   1:  PR[GP1:91,2] = PR[GP1:90,2] + 24.586;
   1:L PR[91] 10mm/sec CNT100;
   1:  PR[GP1:91,1] = PR[GP1:90,1] + 8.241;
   1:  PR[GP1:91,2] = PR[GP1:90,2] + 23.035;
   1:L PR[91] 10mm/sec CNT100;
   1:  PR[GP1:91,1] = PR[GP1:90,1] + 4.572;
   1:  PR[GP1:91,2] = PR[GP1:90,2] + 17.187;
   1:L PR[91] 10mm/sec CNT100;
   1:  PR[GP1:91,1] = PR[GP1:90,1] + 2.350;
   1:  PR[GP1:91,2] = PR[GP1:90,2] + 14.091;
   1:L PR[91] 10mm/sec CNT100;
   1:  PR[GP1:91,1] = PR[GP1:90,1] + -2.900;
   1:L PR[91] 10mm/sec CNT100;
   1:  PR[GP1:91,1] = PR[GP1:90,1] + -6.756;
   1:  PR[GP1:91,2] = PR[GP1:90,2] + 20.165;
   1:L PR[91] 10mm/sec CNT100;
   1:  PR[GP1:91,1] = PR[GP1:90,1] + -8.743;
   1:  PR[GP1:91,2] = PR[GP1:90,2] + 23.019;
   1:L PR[91] 10mm/sec CNT100;
   1:  PR[GP1:91,1] = PR[GP1:90,1] + -10.484;
   1:  PR[GP1:91,2] = PR[GP1:90,2] + 24.588;
   1:L PR[91] 10mm/sec CNT100;
   1:  PR[GP1:91,1] = PR[GP1:90,1] + -18.525;
   1:  PR[GP1:91,2] = PR[GP1:90,2] + 30.630;
   1:L PR[91] 10mm/sec CNT100;
   1:  PR[GP1:91,1] = PR[GP1:90,1] + -19.030;
   1:  PR[GP1:91,2] = PR[GP1:90,2] + 30.917;
   1:L PR[91] 10mm/sec CNT100;
   1:  PR[GP1:91,1] = PR[GP1:90,1] + -21.878;
   1:  PR[GP1:91,2] = PR[GP1:90,2] + 31.816;
   1:L PR[91] 10mm/sec CNT100;
   1:  PR[GP1:91,1] = PR[GP1:90,1] + -30.388;
   1:  PR[GP1:91,2] = PR[GP1:90,2] + 34.743;
   1:L PR[91] 10mm/sec CNT100;
   1:  PR[GP1:91,1] = PR[GP1:90,1] + -33.292;
   1:  PR[GP1:91,2] = PR[GP1:90,2] + 34.868;
   1:L PR[91] 10mm/sec CNT100;
   1:  PR[GP1:91,1] = PR[GP1:90,1] + -42.531;
   1:  PR[GP1:91,2] = PR[GP1:90,2] + 34.793;
   1:L PR[91] 10mm/sec CNT100;
   1:  PR[GP1:91,1] = PR[GP1:90,1] + -48.692;
   1:  PR[GP1:91,2] = PR[GP1:90,2] + 32.836;
   1:L PR[91] 10mm/sec CNT100;
   1:  PR[GP1:91,1] = PR[GP1:90,1] + -54.219;
   1:  PR[GP1:91,2] = PR[GP1:90,2] + 30.834;
   1:L PR[91] 10mm/sec CNT100;
   1:  PR[GP1:91,1] = PR[GP1:90,1] + -61.326;
   1:  PR[GP1:91,2] = PR[GP1:90,2] + 25.314;
   1:L PR[91] 10mm/sec CNT100;
   1:  PR[GP1:91,1] = PR[GP1:90,1] + -63.971;
   1:  PR[GP1:91,2] = PR[GP1:90,2] + 23.133;
   1:L PR[91] 10mm/sec CNT100;
   1:  PR[GP1:91,1] = PR[GP1:90,1] + -69.432;
   1:  PR[GP1:91,2] = PR[GP1:90,2] + 14.214;
   1:L PR[91] 10mm/sec CNT100;
   1:  PR[GP1:91,1] = PR[GP1:90,1] + -70.446;
   1:  PR[GP1:91,2] = PR[GP1:90,2] + 12.486;
   1:L PR[91] 10mm/sec CNT100;
   1:  PR[GP1:91,1] = PR[GP1:90,1] + -72.467;
   1:  PR[GP1:91,2] = PR[GP1:90,2] + 1.672;
   1:L PR[91] 10mm/sec CNT100;
   1:  PR[GP1:91,1] = PR[GP1:90,1] + -72.701;
   1:  PR[GP1:91,2] = PR[GP1:90,2] + 0.583;
   1:L PR[91] 10mm/sec CNT100;
   1:  PR[GP1:91,1] = PR[GP1:90,1] + -72.755;
   1:  PR[GP1:91,2] = PR[GP1:90,2] + 0.282;
   1:L PR[91] 10mm/sec CNT100;
   1:  PR[GP1:91,1] = PR[GP1:90,1] + -70.738;
   1:  PR[GP1:91,2] = PR[GP1:90,2] + -10.290;
   1:L PR[91] 10mm/sec CNT100;
   1:  PR[GP1:91,1] = PR[GP1:90,1] + -70.445;
   1:  PR[GP1:91,2] = PR[GP1:90,2] + -11.930;
   1:L PR[91] 10mm/sec CNT100;
   1:  PR[GP1:91,1] = PR[GP1:90,1] + -69.432;
   1:  PR[GP1:91,2] = PR[GP1:90,2] + -13.656;
   1:L PR[91] 10mm/sec CNT100;
   1:  PR[GP1:91,1] = PR[GP1:90,1] + -63.971;
   1:  PR[GP1:91,2] = PR[GP1:90,2] + -22.575;
   1:L PR[91] 10mm/sec CNT100;
   1:  PR[GP1:91,1] = PR[GP1:90,1] + -61.326;
   1:  PR[GP1:91,2] = PR[GP1:90,2] + -24.756;
   1:L PR[91] 10mm/sec CNT100;
   1:  PR[GP1:91,1] = PR[GP1:90,1] + -54.219;
   1:  PR[GP1:91,2] = PR[GP1:90,2] + -30.276;
   1:L PR[91] 10mm/sec CNT100;
   1:  PR[GP1:91,1] = PR[GP1:90,1] + -48.692;
   1:  PR[GP1:91,2] = PR[GP1:90,2] + -32.278;
   1:L PR[91] 10mm/sec CNT100;
   1:  PR[GP1:91,1] = PR[GP1:90,1] + -42.531;
   1:  PR[GP1:91,2] = PR[GP1:90,2] + -34.235;
   1:L PR[91] 10mm/sec CNT100;
   1:  PR[GP1:91,1] = PR[GP1:90,1] + -33.292;
   1:  PR[GP1:91,2] = PR[GP1:90,2] + -34.310;
   1:L PR[91] 10mm/sec CNT100;
   1:  PR[GP1:91,1] = PR[GP1:90,1] + -30.388;
   1:  PR[GP1:91,2] = PR[GP1:90,2] + -34.185;
   1:L PR[91] 10mm/sec CNT100;
   1:  PR[GP1:91,1] = PR[GP1:90,1] + -21.879;
   1:  PR[GP1:91,2] = PR[GP1:90,2] + -31.258;
   1:L PR[91] 10mm/sec CNT100;
   1:  PR[GP1:91,1] = PR[GP1:90,1] + -19.381;
   1:  PR[GP1:91,2] = PR[GP1:90,2] + -30.458;
   1:L PR[91] 10mm/sec CNT100;
   1:  PR[GP1:91,1] = PR[GP1:90,1] + -19.024;
   1:  PR[GP1:91,2] = PR[GP1:90,2] + -30.355;
   1:L PR[91] 10mm/sec CNT100;
   1:  PR[GP1:91,1] = PR[GP1:90,1] + -18.525;
   1:  PR[GP1:91,2] = PR[GP1:90,2] + -30.072;
   1:L PR[91] 10mm/sec CNT100;
   1:  PR[GP1:91,1] = PR[GP1:90,1] + -10.484;
   1:  PR[GP1:91,2] = PR[GP1:90,2] + -24.030;
   1:L PR[91] 10mm/sec CNT100;
   1:  PR[GP1:91,1] = PR[GP1:90,1] + -8.754;
   1:  PR[GP1:91,2] = PR[GP1:90,2] + -22.471;
   1:L PR[91] 10mm/sec CNT100;
   1:  PR[GP1:91,1] = PR[GP1:90,1] + -5.085;
   1:  PR[GP1:91,2] = PR[GP1:90,2] + -16.617;
   1:L PR[91] 10mm/sec CNT100;
   1:  PR[GP1:91,1] = PR[GP1:90,1] + -2.878;
   1:  PR[GP1:91,2] = PR[GP1:90,2] + -13.533;
   1:L PR[91] 10mm/sec CNT100;
   1:  PR[GP1:91,1] = PR[GP1:90,1] + 2.371;
   1:L PR[91] 10mm/sec CNT100;
   1:  PR[GP1:91,1] = PR[GP1:90,1] + 5.458;
   1:  PR[GP1:91,2] = PR[GP1:90,2] + -18.880;
   1:  PR[GP1:91,3] = PR[GP1:90,3] + 33.855;
   1:L PR[91] 10mm/sec CNT100;
   1:  PR[GP1:91,1] = PR[GP1:90,1] + 7.960;
   1:  PR[GP1:91,2] = PR[GP1:90,2] + -22.465;
   1:L PR[91] 10mm/sec CNT100;
   1:  PR[GP1:91,1] = PR[GP1:90,1] + 10.133;
   1:  PR[GP1:91,2] = PR[GP1:90,2] + -24.423;
   1:L PR[91] 10mm/sec CNT100;
   1:  PR[GP1:91,1] = PR[GP1:90,1] + 17.353;
   1:  PR[GP1:91,2] = PR[GP1:90,2] + -29.858;
   1:L PR[91] 10mm/sec CNT100;
   1:  PR[GP1:91,1] = PR[GP1:90,1] + 18.470;
   1:  PR[GP1:91,2] = PR[GP1:90,2] + -30.491;
   1:L PR[91] 10mm/sec CNT100;
   1:  PR[GP1:91,1] = PR[GP1:90,1] + 24.347;
   1:  PR[GP1:91,2] = PR[GP1:90,2] + -32.346;
   1:L PR[91] 10mm/sec CNT100;
   1:  PR[GP1:91,1] = PR[GP1:90,1] + 29.865;
   1:  PR[GP1:91,2] = PR[GP1:90,2] + -34.244;
   1:L PR[91] 10mm/sec CNT100;
   1:  PR[GP1:91,1] = PR[GP1:90,1] + 31.722;
   1:  PR[GP1:91,2] = PR[GP1:90,2] + -34.324;
   1:L PR[91] 10mm/sec CNT100;
   1:  PR[GP1:91,1] = PR[GP1:90,1] + 41.979;
   1:  PR[GP1:91,2] = PR[GP1:90,2] + -34.242;
   1:L PR[91] 10mm/sec CNT100;
   1:  PR[GP1:91,1] = PR[GP1:90,1] + 47.240;
   1:  PR[GP1:91,2] = PR[GP1:90,2] + -32.573;
   1:L PR[91] 10mm/sec CNT100;
   1:  PR[GP1:91,1] = PR[GP1:90,1] + 53.633;
   1:  PR[GP1:91,2] = PR[GP1:90,2] + -30.260;
   1:L PR[91] 10mm/sec CNT100;
   1:  PR[GP1:91,1] = PR[GP1:90,1] + 60.074;
   1:  PR[GP1:91,2] = PR[GP1:90,2] + -25.257;
   1:L PR[91] 10mm/sec CNT100;
   1:  PR[GP1:91,1] = PR[GP1:90,1] + 63.355;
   1:  PR[GP1:91,2] = PR[GP1:90,2] + -22.547;
   1:L PR[91] 10mm/sec CNT100;
   1:  PR[GP1:91,1] = PR[GP1:90,1] + 68.421;
   1:  PR[GP1:91,2] = PR[GP1:90,2] + -14.287;
   1:L PR[91] 10mm/sec CNT100;
   1:  PR[GP1:91,1] = PR[GP1:90,1] + 69.810;
   1:  PR[GP1:91,2] = PR[GP1:90,2] + -11.926;
   1:L PR[91] 10mm/sec CNT100;
   1:  PR[GP1:91,1] = PR[GP1:90,1] + 71.704;
   1:  PR[GP1:91,2] = PR[GP1:90,2] + -1.787;
   1:L PR[91] 10mm/sec CNT100;
   1:  PR[GP1:91,1] = PR[GP1:90,1] + 71.924;
   1:  PR[GP1:91,2] = PR[GP1:90,2] + -0.764;
   1:L PR[91] 10mm/sec CNT100;
   1:  PR[GP1:91,1] = PR[GP1:90,1] + 72.110;
   1:  PR[GP1:91,2] = PR[GP1:90,2] + 0.276;
   1:L PR[91] 10mm/sec CNT100;
   1:  PR[GP1:91,1] = PR[GP1:90,1] + 70.212;
   1:  PR[GP1:91,2] = PR[GP1:90,2] + 10.230;
   1:L PR[91] 10mm/sec CNT100;
   1:  PR[GP1:91,1] = PR[GP1:90,1] + 69.809;
   1:  PR[GP1:91,2] = PR[GP1:90,2] + 12.486;
   1:L PR[91] 10mm/sec CNT100;
   1:  PR[GP1:91,1] = PR[GP1:90,1] + 68.421;
   1:  PR[GP1:91,2] = PR[GP1:90,2] + 14.845;
   1:L PR[91] 10mm/sec CNT100;
   1:  PR[GP1:91,1] = PR[GP1:90,1] + 63.355;
   1:  PR[GP1:91,2] = PR[GP1:90,2] + 23.106;
   1:L PR[91] 10mm/sec CNT100;
   1:  PR[GP1:91,1] = PR[GP1:90,1] + 60.074;
   1:  PR[GP1:91,2] = PR[GP1:90,2] + 25.815;
   1:L PR[91] 10mm/sec CNT100;
   1:  PR[GP1:91,1] = PR[GP1:90,1] + 53.633;
   1:  PR[GP1:91,2] = PR[GP1:90,2] + 30.818;
   1:L PR[91] 10mm/sec CNT100;
   1:  PR[GP1:91,1] = PR[GP1:90,1] + 47.240;
   1:  PR[GP1:91,2] = PR[GP1:90,2] + 33.131;
   1:L PR[91] 10mm/sec CNT100;
   1:  PR[GP1:91,1] = PR[GP1:90,1] + 41.979;
   1:  PR[GP1:91,2] = PR[GP1:90,2] + 34.800;
   1:L PR[91] 10mm/sec CNT100;
   1:  PR[GP1:91,1] = PR[GP1:90,1] + 31.722;
   1:  PR[GP1:91,2] = PR[GP1:90,2] + 34.882;
   1:L PR[91] 10mm/sec CNT100;
   1:  PR[GP1:91,1] = PR[GP1:90,1] + 29.865;
   1:  PR[GP1:91,2] = PR[GP1:90,2] + 34.802;
   1:L PR[91] 10mm/sec CNT100;
   1:  PR[GP1:91,1] = PR[GP1:90,1] + 24.348;
   1:  PR[GP1:91,2] = PR[GP1:90,2] + 32.905;
   1:L PR[91] 10mm/sec CNT100;
   1:  PR[GP1:91,1] = PR[GP1:90,1] + 19.257;
   1:  PR[GP1:91,2] = PR[GP1:90,2] + 31.274;
   1:L PR[91] 10mm/sec CNT100;
   1:  PR[GP1:91,1] = PR[GP1:90,1] + 18.464;
   1:  PR[GP1:91,2] = PR[GP1:90,2] + 31.045;
   1:L PR[91] 10mm/sec CNT100;
   1:  PR[GP1:91,1] = PR[GP1:90,1] + 17.353;
   1:  PR[GP1:91,2] = PR[GP1:90,2] + 30.416;
   1:L PR[91] 10mm/sec CNT100;
   1:  PR[GP1:91,1] = PR[GP1:90,1] + 10.133;
   1:  PR[GP1:91,2] = PR[GP1:90,2] + 24.981;
   1:L PR[91] 10mm/sec CNT100;
   1:  PR[GP1:91,1] = PR[GP1:90,1] + 7.971;
   1:  PR[GP1:91,2] = PR[GP1:90,2] + 23.034;
   1:L PR[91] 10mm/sec CNT100;
   1:  PR[GP1:91,1] = PR[GP1:90,1] + 4.797;
   1:  PR[GP1:91,2] = PR[GP1:90,2] + 17.974;
   1:L PR[91] 10mm/sec CNT100;
   1:  PR[GP1:91,1] = PR[GP1:90,1] + 2.243;
   1:  PR[GP1:91,2] = PR[GP1:90,2] + 14.416;
   1:L PR[91] 10mm/sec CNT100;
   1:  PR[GP1:91,1] = PR[GP1:90,1] + -2.792;
   1:L PR[91] 10mm/sec CNT100;
   1:  PR[GP1:91,1] = PR[GP1:90,1] + -5.985;
   1:  PR[GP1:91,2] = PR[GP1:90,2] + 19.445;
   1:L PR[91] 10mm/sec CNT100;
   1:  PR[GP1:91,1] = PR[GP1:90,1] + -8.469;
   1:  PR[GP1:91,2] = PR[GP1:90,2] + 23.013;
   1:L PR[91] 10mm/sec CNT100;
   1:  PR[GP1:91,1] = PR[GP1:90,1] + -10.652;
   1:  PR[GP1:91,2] = PR[GP1:90,2] + 24.980;
   1:L PR[91] 10mm/sec CNT100;
   1:  PR[GP1:91,1] = PR[GP1:90,1] + -17.878;
   1:  PR[GP1:91,2] = PR[GP1:90,2] + 30.410;
   1:L PR[91] 10mm/sec CNT100;
   1:  PR[GP1:91,1] = PR[GP1:90,1] + -19.003;
   1:  PR[GP1:91,2] = PR[GP1:90,2] + 31.049;
   1:L PR[91] 10mm/sec CNT100;
   1:  PR[GP1:91,1] = PR[GP1:90,1] + -24.873;
   1:  PR[GP1:91,2] = PR[GP1:90,2] + 32.903;
   1:L PR[91] 10mm/sec CNT100;
   1:  PR[GP1:91,1] = PR[GP1:90,1] + -30.398;
   1:  PR[GP1:91,2] = PR[GP1:90,2] + 34.803;
   1:L PR[91] 10mm/sec CNT100;
   1:  PR[GP1:91,1] = PR[GP1:90,1] + -32.256;
   1:  PR[GP1:91,2] = PR[GP1:90,2] + 34.883;
   1:L PR[91] 10mm/sec CNT100;
   1:  PR[GP1:91,1] = PR[GP1:90,1] + -42.512;
   1:  PR[GP1:91,2] = PR[GP1:90,2] + 34.799;
   1:L PR[91] 10mm/sec CNT100;
   1:  PR[GP1:91,1] = PR[GP1:90,1] + -47.772;
   1:  PR[GP1:91,2] = PR[GP1:90,2] + 33.129;
   1:L PR[91] 10mm/sec CNT100;
   1:  PR[GP1:91,1] = PR[GP1:90,1] + -54.165;
   1:  PR[GP1:91,2] = PR[GP1:90,2] + 30.814;
   1:L PR[91] 10mm/sec CNT100;
   1:  PR[GP1:91,1] = PR[GP1:90,1] + -60.604;
   1:  PR[GP1:91,2] = PR[GP1:90,2] + 25.812;
   1:L PR[91] 10mm/sec CNT100;
   1:  PR[GP1:91,1] = PR[GP1:90,1] + -63.884;
   1:  PR[GP1:91,2] = PR[GP1:90,2] + 23.107;
   1:L PR[91] 10mm/sec CNT100;
   1:  PR[GP1:91,1] = PR[GP1:90,1] + -68.948;
   1:  PR[GP1:91,2] = PR[GP1:90,2] + 14.837;
   1:L PR[91] 10mm/sec CNT100;
   1:  PR[GP1:91,1] = PR[GP1:90,1] + -70.338;
   1:  PR[GP1:91,2] = PR[GP1:90,2] + 12.469;
   1:L PR[91] 10mm/sec CNT100;
   1:  PR[GP1:91,1] = PR[GP1:90,1] + -72.230;
   1:  PR[GP1:91,2] = PR[GP1:90,2] + 2.341;
   1:L PR[91] 10mm/sec CNT100;
   1:  PR[GP1:91,1] = PR[GP1:90,1] + -72.450;
   1:  PR[GP1:91,2] = PR[GP1:90,2] + 1.320;
   1:L PR[91] 10mm/sec CNT100;
   1:  PR[GP1:91,1] = PR[GP1:90,1] + -72.636;
   1:  PR[GP1:91,2] = PR[GP1:90,2] + 0.282;
   1:L PR[91] 10mm/sec CNT100;
   1:  PR[GP1:91,1] = PR[GP1:90,1] + -70.739;
   1:  PR[GP1:91,2] = PR[GP1:90,2] + -9.661;
   1:L PR[91] 10mm/sec CNT100;
   1:  PR[GP1:91,1] = PR[GP1:90,1] + -70.336;
   1:  PR[GP1:91,2] = PR[GP1:90,2] + -11.913;
   1:L PR[91] 10mm/sec CNT100;
   1:  PR[GP1:91,1] = PR[GP1:90,1] + -68.948;
   1:  PR[GP1:91,2] = PR[GP1:90,2] + -14.279;
   1:L PR[91] 10mm/sec CNT100;
   1:  PR[GP1:91,1] = PR[GP1:90,1] + -63.884;
   1:  PR[GP1:91,2] = PR[GP1:90,2] + -22.549;
   1:L PR[91] 10mm/sec CNT100;
   1:  PR[GP1:91,1] = PR[GP1:90,1] + -60.604;
   1:  PR[GP1:91,2] = PR[GP1:90,2] + -25.254;
   1:L PR[91] 10mm/sec CNT100;
   1:  PR[GP1:91,1] = PR[GP1:90,1] + -54.165;
   1:  PR[GP1:91,2] = PR[GP1:90,2] + -30.256;
   1:L PR[91] 10mm/sec CNT100;
   1:  PR[GP1:91,1] = PR[GP1:90,1] + -47.772;
   1:  PR[GP1:91,2] = PR[GP1:90,2] + -32.570;
   1:L PR[91] 10mm/sec CNT100;
   1:  PR[GP1:91,1] = PR[GP1:90,1] + -42.512;
   1:  PR[GP1:91,2] = PR[GP1:90,2] + -34.241;
   1:L PR[91] 10mm/sec CNT100;
   1:  PR[GP1:91,1] = PR[GP1:90,1] + -32.256;
   1:  PR[GP1:91,2] = PR[GP1:90,2] + -34.325;
   1:L PR[91] 10mm/sec CNT100;
   1:  PR[GP1:91,1] = PR[GP1:90,1] + -30.398;
   1:  PR[GP1:91,2] = PR[GP1:90,2] + -34.245;
   1:L PR[91] 10mm/sec CNT100;
   1:  PR[GP1:91,1] = PR[GP1:90,1] + -24.874;
   1:  PR[GP1:91,2] = PR[GP1:90,2] + -32.345;
   1:L PR[91] 10mm/sec CNT100;
   1:  PR[GP1:91,1] = PR[GP1:90,1] + -19.788;
   1:  PR[GP1:91,2] = PR[GP1:90,2] + -30.716;
   1:L PR[91] 10mm/sec CNT100;
   1:  PR[GP1:91,1] = PR[GP1:90,1] + -18.997;
   1:  PR[GP1:91,2] = PR[GP1:90,2] + -30.488;
   1:L PR[91] 10mm/sec CNT100;
   1:  PR[GP1:91,1] = PR[GP1:90,1] + -17.878;
   1:  PR[GP1:91,2] = PR[GP1:90,2] + -29.852;
   1:L PR[91] 10mm/sec CNT100;
   1:  PR[GP1:91,1] = PR[GP1:90,1] + -10.652;
   1:  PR[GP1:91,2] = PR[GP1:90,2] + -24.422;
   1:L PR[91] 10mm/sec CNT100;
   1:  PR[GP1:91,1] = PR[GP1:90,1] + -8.480;
   1:  PR[GP1:91,2] = PR[GP1:90,2] + -22.465;
   1:L PR[91] 10mm/sec CNT100;
   1:  PR[GP1:91,1] = PR[GP1:90,1] + -5.306;
   1:  PR[GP1:91,2] = PR[GP1:90,2] + -17.402;
   1:L PR[91] 10mm/sec CNT100;
   1:  PR[GP1:91,1] = PR[GP1:90,1] + -2.770;
   1:  PR[GP1:91,2] = PR[GP1:90,2] + -13.858;
   1:L PR[91] 10mm/sec CNT100;
   1:  PR[GP1:91,1] = PR[GP1:90,1] + 2.264;
   1:L PR[91] 10mm/sec CNT100;
   1:  PR[GP1:91,1] = PR[GP1:90,1] + 4.688;
   1:  PR[GP1:91,2] = PR[GP1:90,2] + -18.162;
   1:  PR[GP1:91,3] = PR[GP1:90,3] + 34.465;
   1:L PR[91] 10mm/sec CNT100;
   1:  PR[GP1:91,1] = PR[GP1:90,1] + 7.690;
   1:  PR[GP1:91,2] = PR[GP1:90,2] + -22.464;
   1:L PR[91] 10mm/sec CNT100;
   1:  PR[GP1:91,1] = PR[GP1:90,1] + 10.303;
   1:  PR[GP1:91,2] = PR[GP1:90,2] + -24.818;
   1:L PR[91] 10mm/sec CNT100;
   1:  PR[GP1:91,1] = PR[GP1:90,1] + 16.711;
   1:  PR[GP1:91,2] = PR[GP1:90,2] + -29.642;
   1:L PR[91] 10mm/sec CNT100;
   1:  PR[GP1:91,1] = PR[GP1:90,1] + 18.443;
   1:  PR[GP1:91,2] = PR[GP1:90,2] + -30.623;
   1:L PR[91] 10mm/sec CNT100;
   1:  PR[GP1:91,1] = PR[GP1:90,1] + 27.342;
   1:  PR[GP1:91,2] = PR[GP1:90,2] + -33.433;
   1:L PR[91] 10mm/sec CNT100;
   1:  PR[GP1:91,1] = PR[GP1:90,1] + 29.876;
   1:  PR[GP1:91,2] = PR[GP1:90,2] + -34.304;
   1:L PR[91] 10mm/sec CNT100;
   1:  PR[GP1:91,1] = PR[GP1:90,1] + 30.687;
   1:  PR[GP1:91,2] = PR[GP1:90,2] + -34.339;
   1:L PR[91] 10mm/sec CNT100;
   1:  PR[GP1:91,1] = PR[GP1:90,1] + 41.960;
   1:  PR[GP1:91,2] = PR[GP1:90,2] + -34.249;
   1:L PR[91] 10mm/sec CNT100;
   1:  PR[GP1:91,1] = PR[GP1:90,1] + 46.320;
   1:  PR[GP1:91,2] = PR[GP1:90,2] + -32.866;
   1:L PR[91] 10mm/sec CNT100;
   1:  PR[GP1:91,1] = PR[GP1:90,1] + 53.579;
   1:  PR[GP1:91,2] = PR[GP1:90,2] + -30.240;
   1:L PR[91] 10mm/sec CNT100;
   1:  PR[GP1:91,1] = PR[GP1:90,1] + 59.352;
   1:  PR[GP1:91,2] = PR[GP1:90,2] + -25.755;
   1:L PR[91] 10mm/sec CNT100;
   1:  PR[GP1:91,1] = PR[GP1:90,1] + 63.269;
   1:  PR[GP1:91,2] = PR[GP1:90,2] + -22.521;
   1:L PR[91] 10mm/sec CNT100;
   1:  PR[GP1:91,1] = PR[GP1:90,1] + 67.937;
   1:  PR[GP1:91,2] = PR[GP1:90,2] + -14.909;
   1:L PR[91] 10mm/sec CNT100;
   1:  PR[GP1:91,1] = PR[GP1:90,1] + 69.702;
   1:  PR[GP1:91,2] = PR[GP1:90,2] + -11.909;
   1:L PR[91] 10mm/sec CNT100;
   1:  PR[GP1:91,1] = PR[GP1:90,1] + 71.467;
   1:  PR[GP1:91,2] = PR[GP1:90,2] + -2.457;
   1:L PR[91] 10mm/sec CNT100;
   1:  PR[GP1:91,1] = PR[GP1:90,1] + 71.672;
   1:  PR[GP1:91,2] = PR[GP1:90,2] + -1.503;
   1:L PR[91] 10mm/sec CNT100;
   1:  PR[GP1:91,1] = PR[GP1:90,1] + 71.991;
   1:  PR[GP1:91,2] = PR[GP1:90,2] + 0.276;
   1:L PR[91] 10mm/sec CNT100;
   1:  PR[GP1:91,1] = PR[GP1:90,1] + 70.212;
   1:  PR[GP1:91,2] = PR[GP1:90,2] + 9.601;
   1:L PR[91] 10mm/sec CNT100;
   1:  PR[GP1:91,1] = PR[GP1:90,1] + 69.701;
   1:  PR[GP1:91,2] = PR[GP1:90,2] + 12.469;
   1:L PR[91] 10mm/sec CNT100;
   1:  PR[GP1:91,1] = PR[GP1:90,1] + 67.937;
   1:  PR[GP1:91,2] = PR[GP1:90,2] + 15.467;
   1:L PR[91] 10mm/sec CNT100;
   1:  PR[GP1:91,1] = PR[GP1:90,1] + 63.269;
   1:  PR[GP1:91,2] = PR[GP1:90,2] + 23.079;
   1:L PR[91] 10mm/sec CNT100;
   1:  PR[GP1:91,1] = PR[GP1:90,1] + 59.352;
   1:  PR[GP1:91,2] = PR[GP1:90,2] + 26.313;
   1:L PR[91] 10mm/sec CNT100;
   1:  PR[GP1:91,1] = PR[GP1:90,1] + 53.579;
   1:  PR[GP1:91,2] = PR[GP1:90,2] + 30.798;
   1:L PR[91] 10mm/sec CNT100;
   1:  PR[GP1:91,1] = PR[GP1:90,1] + 46.320;
   1:  PR[GP1:91,2] = PR[GP1:90,2] + 33.424;
   1:L PR[91] 10mm/sec CNT100;
   1:  PR[GP1:91,1] = PR[GP1:90,1] + 41.960;
   1:  PR[GP1:91,2] = PR[GP1:90,2] + 34.807;
   1:L PR[91] 10mm/sec CNT100;
   1:  PR[GP1:91,1] = PR[GP1:90,1] + 30.687;
   1:  PR[GP1:91,2] = PR[GP1:90,2] + 34.897;
   1:L PR[91] 10mm/sec CNT100;
   1:  PR[GP1:91,1] = PR[GP1:90,1] + 29.876;
   1:  PR[GP1:91,2] = PR[GP1:90,2] + 34.862;
   1:L PR[91] 10mm/sec CNT100;
   1:  PR[GP1:91,1] = PR[GP1:90,1] + 27.343;
   1:  PR[GP1:91,2] = PR[GP1:90,2] + 33.991;
   1:L PR[91] 10mm/sec CNT100;
   1:  PR[GP1:91,1] = PR[GP1:90,1] + 19.664;
   1:  PR[GP1:91,2] = PR[GP1:90,2] + 31.531;
   1:L PR[91] 10mm/sec CNT100;
   1:  PR[GP1:91,1] = PR[GP1:90,1] + 18.436;
   1:  PR[GP1:91,2] = PR[GP1:90,2] + 31.177;
   1:L PR[91] 10mm/sec CNT100;
   1:  PR[GP1:91,1] = PR[GP1:90,1] + 16.711;
   1:  PR[GP1:91,2] = PR[GP1:90,2] + 30.200;
   1:L PR[91] 10mm/sec CNT100;
   1:  PR[GP1:91,1] = PR[GP1:90,1] + 10.303;
   1:  PR[GP1:91,2] = PR[GP1:90,2] + 25.376;
   1:L PR[91] 10mm/sec CNT100;
   1:  PR[GP1:91,1] = PR[GP1:90,1] + 7.702;
   1:  PR[GP1:91,2] = PR[GP1:90,2] + 23.032;
   1:L PR[91] 10mm/sec CNT100;
   1:  PR[GP1:91,1] = PR[GP1:90,1] + 5.022;
   1:  PR[GP1:91,2] = PR[GP1:90,2] + 18.762;
   1:L PR[91] 10mm/sec CNT100;
   1:  PR[GP1:91,1] = PR[GP1:90,1] + 2.136;
   1:  PR[GP1:91,2] = PR[GP1:90,2] + 14.741;
   1:L PR[91] 10mm/sec CNT100;
   1:  PR[GP1:91,1] = PR[GP1:90,1] + -2.684;
   1:L PR[91] 10mm/sec CNT100;
   1:  PR[GP1:91,1] = PR[GP1:90,1] + -5.214;
   1:  PR[GP1:91,2] = PR[GP1:90,2] + 18.725;
   1:L PR[91] 10mm/sec CNT100;
   1:  PR[GP1:91,1] = PR[GP1:90,1] + -8.194;
   1:  PR[GP1:91,2] = PR[GP1:90,2] + 23.007;
   1:L PR[91] 10mm/sec CNT100;
   1:  PR[GP1:91,1] = PR[GP1:90,1] + -10.819;
   1:  PR[GP1:91,2] = PR[GP1:90,2] + 25.372;
   1:L PR[91] 10mm/sec CNT100;
   1:  PR[GP1:91,1] = PR[GP1:90,1] + -17.232;
   1:  PR[GP1:91,2] = PR[GP1:90,2] + 30.191;
   1:L PR[91] 10mm/sec CNT100;
   1:  PR[GP1:91,1] = PR[GP1:90,1] + -18.976;
   1:  PR[GP1:91,2] = PR[GP1:90,2] + 31.182;
   1:L PR[91] 10mm/sec CNT100;
   1:  PR[GP1:91,1] = PR[GP1:90,1] + -27.868;
   1:  PR[GP1:91,2] = PR[GP1:90,2] + 33.989;
   1:L PR[91] 10mm/sec CNT100;
   1:  PR[GP1:91,1] = PR[GP1:90,1] + -30.408;
   1:  PR[GP1:91,2] = PR[GP1:90,2] + 34.863;
   1:L PR[91] 10mm/sec CNT100;
   1:  PR[GP1:91,1] = PR[GP1:90,1] + -31.221;
   1:  PR[GP1:91,2] = PR[GP1:90,2] + 34.898;
   1:L PR[91] 10mm/sec CNT100;
   1:  PR[GP1:91,1] = PR[GP1:90,1] + -42.493;
   1:  PR[GP1:91,2] = PR[GP1:90,2] + 34.806;
   1:L PR[91] 10mm/sec CNT100;
   1:  PR[GP1:91,1] = PR[GP1:90,1] + -46.853;
   1:  PR[GP1:91,2] = PR[GP1:90,2] + 33.421;
   1:L PR[91] 10mm/sec CNT100;
   1:  PR[GP1:91,1] = PR[GP1:90,1] + -54.110;
   1:  PR[GP1:91,2] = PR[GP1:90,2] + 30.793;
   1:L PR[91] 10mm/sec CNT100;
   1:  PR[GP1:91,1] = PR[GP1:90,1] + -59.882;
   1:  PR[GP1:91,2] = PR[GP1:90,2] + 26.310;
   1:L PR[91] 10mm/sec CNT100;
   1:  PR[GP1:91,1] = PR[GP1:90,1] + -63.798;
   1:  PR[GP1:91,2] = PR[GP1:90,2] + 23.082;
   1:L PR[91] 10mm/sec CNT100;
   1:  PR[GP1:91,1] = PR[GP1:90,1] + -68.464;
   1:  PR[GP1:91,2] = PR[GP1:90,2] + 15.460;
   1:L PR[91] 10mm/sec CNT100;
   1:  PR[GP1:91,1] = PR[GP1:90,1] + -70.229;
   1:  PR[GP1:91,2] = PR[GP1:90,2] + 12.452;
   1:L PR[91] 10mm/sec CNT100;
   1:  PR[GP1:91,1] = PR[GP1:90,1] + -71.993;
   1:  PR[GP1:91,2] = PR[GP1:90,2] + 3.010;
   1:L PR[91] 10mm/sec CNT100;
   1:  PR[GP1:91,1] = PR[GP1:90,1] + -72.199;
   1:  PR[GP1:91,2] = PR[GP1:90,2] + 2.058;
   1:L PR[91] 10mm/sec CNT100;
   1:  PR[GP1:91,1] = PR[GP1:90,1] + -72.517;
   1:  PR[GP1:91,2] = PR[GP1:90,2] + 0.282;
   1:L PR[91] 10mm/sec CNT100;
   1:  PR[GP1:91,1] = PR[GP1:90,1] + -70.739;
   1:  PR[GP1:91,2] = PR[GP1:90,2] + -9.033;
   1:L PR[91] 10mm/sec CNT100;
   1:  PR[GP1:91,1] = PR[GP1:90,1] + -70.228;
   1:  PR[GP1:91,2] = PR[GP1:90,2] + -11.896;
   1:L PR[91] 10mm/sec CNT100;
   1:  PR[GP1:91,1] = PR[GP1:90,1] + -68.464;
   1:  PR[GP1:91,2] = PR[GP1:90,2] + -14.903;
   1:L PR[91] 10mm/sec CNT100;
   1:  PR[GP1:91,1] = PR[GP1:90,1] + -63.798;
   1:  PR[GP1:91,2] = PR[GP1:90,2] + -22.524;
   1:L PR[91] 10mm/sec CNT100;
   1:  PR[GP1:91,1] = PR[GP1:90,1] + -59.882;
   1:  PR[GP1:91,2] = PR[GP1:90,2] + -25.752;
   1:L PR[91] 10mm/sec CNT100;
   1:  PR[GP1:91,1] = PR[GP1:90,1] + -54.110;
   1:  PR[GP1:91,2] = PR[GP1:90,2] + -30.235;
   1:L PR[91] 10mm/sec CNT100;
   1:  PR[GP1:91,1] = PR[GP1:90,1] + -46.853;
   1:  PR[GP1:91,2] = PR[GP1:90,2] + -32.863;
   1:L PR[91] 10mm/sec CNT100;
   1:  PR[GP1:91,1] = PR[GP1:90,1] + -42.493;
   1:  PR[GP1:91,2] = PR[GP1:90,2] + -34.248;
   1:L PR[91] 10mm/sec CNT100;
   1:  PR[GP1:91,1] = PR[GP1:90,1] + -31.221;
   1:  PR[GP1:91,2] = PR[GP1:90,2] + -34.340;
   1:L PR[91] 10mm/sec CNT100;
   1:  PR[GP1:91,1] = PR[GP1:90,1] + -30.408;
   1:  PR[GP1:91,2] = PR[GP1:90,2] + -34.305;
   1:L PR[91] 10mm/sec CNT100;
   1:  PR[GP1:91,1] = PR[GP1:90,1] + -27.869;
   1:  PR[GP1:91,2] = PR[GP1:90,2] + -33.432;
   1:L PR[91] 10mm/sec CNT100;
   1:  PR[GP1:91,1] = PR[GP1:90,1] + -20.195;
   1:  PR[GP1:91,2] = PR[GP1:90,2] + -30.973;
   1:L PR[91] 10mm/sec CNT100;
   1:  PR[GP1:91,1] = PR[GP1:90,1] + -18.969;
   1:  PR[GP1:91,2] = PR[GP1:90,2] + -30.620;
   1:L PR[91] 10mm/sec CNT100;
   1:  PR[GP1:91,1] = PR[GP1:90,1] + -17.232;
   1:  PR[GP1:91,2] = PR[GP1:90,2] + -29.633;
   1:L PR[91] 10mm/sec CNT100;
   1:  PR[GP1:91,1] = PR[GP1:90,1] + -10.820;
   1:  PR[GP1:91,2] = PR[GP1:90,2] + -24.814;
   1:L PR[91] 10mm/sec CNT100;
   1:  PR[GP1:91,1] = PR[GP1:90,1] + -8.205;
   1:  PR[GP1:91,2] = PR[GP1:90,2] + -22.459;
   1:L PR[91] 10mm/sec CNT100;
   1:  PR[GP1:91,1] = PR[GP1:90,1] + -5.528;
   1:  PR[GP1:91,2] = PR[GP1:90,2] + -18.187;
   1:L PR[91] 10mm/sec CNT100;
   1:  PR[GP1:91,1] = PR[GP1:90,1] + -2.663;
   1:  PR[GP1:91,2] = PR[GP1:90,2] + -14.183;
   1:L PR[91] 10mm/sec CNT100;
   1:  PR[GP1:91,1] = PR[GP1:90,1] + 2.158;
   1:L PR[91] 10mm/sec CNT100;
   1:  PR[GP1:91,1] = PR[GP1:90,1] + 3.918;
   1:  PR[GP1:91,2] = PR[GP1:90,2] + -17.444;
   1:  PR[GP1:91,3] = PR[GP1:90,3] + 35.075;
   1:L PR[91] 10mm/sec CNT100;
   1:  PR[GP1:91,1] = PR[GP1:90,1] + 7.421;
   1:  PR[GP1:91,2] = PR[GP1:90,2] + -22.463;
   1:L PR[91] 10mm/sec CNT100;
   1:  PR[GP1:91,1] = PR[GP1:90,1] + 10.473;
   1:  PR[GP1:91,2] = PR[GP1:90,2] + -25.213;
   1:L PR[91] 10mm/sec CNT100;
   1:  PR[GP1:91,1] = PR[GP1:90,1] + 16.069;
   1:  PR[GP1:91,2] = PR[GP1:90,2] + -29.425;
   1:L PR[91] 10mm/sec CNT100;
   1:  PR[GP1:91,1] = PR[GP1:90,1] + 18.415;
   1:  PR[GP1:91,2] = PR[GP1:90,2] + -30.755;
   1:L PR[91] 10mm/sec CNT100;
   1:  PR[GP1:91,1] = PR[GP1:90,1] + 29.819;
   1:  PR[GP1:91,2] = PR[GP1:90,2] + -34.354;
   1:L PR[91] 10mm/sec CNT100;
   1:  PR[GP1:91,1] = PR[GP1:90,1] + 41.942;
   1:  PR[GP1:91,2] = PR[GP1:90,2] + -34.256;
   1:L PR[91] 10mm/sec CNT100;
   1:  PR[GP1:91,1] = PR[GP1:90,1] + 45.401;
   1:  PR[GP1:91,2] = PR[GP1:90,2] + -33.158;
   1:L PR[91] 10mm/sec CNT100;
   1:  PR[GP1:91,1] = PR[GP1:90,1] + 53.525;
   1:  PR[GP1:91,2] = PR[GP1:90,2] + -30.220;
   1:L PR[91] 10mm/sec CNT100;
   1:  PR[GP1:91,1] = PR[GP1:90,1] + 58.630;
   1:  PR[GP1:91,2] = PR[GP1:90,2] + -26.253;
   1:L PR[91] 10mm/sec CNT100;
   1:  PR[GP1:91,1] = PR[GP1:90,1] + 63.182;
   1:  PR[GP1:91,2] = PR[GP1:90,2] + -22.495;
   1:L PR[91] 10mm/sec CNT100;
   1:  PR[GP1:91,1] = PR[GP1:90,1] + 67.453;
   1:  PR[GP1:91,2] = PR[GP1:90,2] + -15.531;
   1:L PR[91] 10mm/sec CNT100;
   1:  PR[GP1:91,1] = PR[GP1:90,1] + 69.593;
   1:  PR[GP1:91,2] = PR[GP1:90,2] + -11.893;
   1:L PR[91] 10mm/sec CNT100;
   1:  PR[GP1:91,1] = PR[GP1:90,1] + 71.230;
   1:  PR[GP1:91,2] = PR[GP1:90,2] + -3.127;
   1:L PR[91] 10mm/sec CNT100;
   1:  PR[GP1:91,1] = PR[GP1:90,1] + 71.421;
   1:  PR[GP1:91,2] = PR[GP1:90,2] + -2.241;
   1:L PR[91] 10mm/sec CNT100;
   1:  PR[GP1:91,1] = PR[GP1:90,1] + 71.871;
   1:  PR[GP1:91,2] = PR[GP1:90,2] + 0.276;
   1:L PR[91] 10mm/sec CNT100;
   1:  PR[GP1:91,1] = PR[GP1:90,1] + 70.213;
   1:  PR[GP1:91,2] = PR[GP1:90,2] + 8.972;
   1:L PR[91] 10mm/sec CNT100;
   1:  PR[GP1:91,1] = PR[GP1:90,1] + 69.592;
   1:  PR[GP1:91,2] = PR[GP1:90,2] + 12.453;
   1:L PR[91] 10mm/sec CNT100;
   1:  PR[GP1:91,1] = PR[GP1:90,1] + 67.453;
   1:  PR[GP1:91,2] = PR[GP1:90,2] + 16.089;
   1:L PR[91] 10mm/sec CNT100;
   1:  PR[GP1:91,1] = PR[GP1:90,1] + 63.182;
   1:  PR[GP1:91,2] = PR[GP1:90,2] + 23.053;
   1:L PR[91] 10mm/sec CNT100;
   1:  PR[GP1:91,1] = PR[GP1:90,1] + 58.630;
   1:  PR[GP1:91,2] = PR[GP1:90,2] + 26.811;
   1:L PR[91] 10mm/sec CNT100;
   1:  PR[GP1:91,1] = PR[GP1:90,1] + 53.525;
   1:  PR[GP1:91,2] = PR[GP1:90,2] + 30.778;
   1:L PR[91] 10mm/sec CNT100;
   1:  PR[GP1:91,1] = PR[GP1:90,1] + 45.401;
   1:  PR[GP1:91,2] = PR[GP1:90,2] + 33.716;
   1:L PR[91] 10mm/sec CNT100;
   1:  PR[GP1:91,1] = PR[GP1:90,1] + 41.942;
   1:  PR[GP1:91,2] = PR[GP1:90,2] + 34.814;
   1:L PR[91] 10mm/sec CNT100;
   1:  PR[GP1:91,1] = PR[GP1:90,1] + 29.821;
   1:  PR[GP1:91,2] = PR[GP1:90,2] + 34.912;
   1:L PR[91] 10mm/sec CNT100;
   1:  PR[GP1:91,1] = PR[GP1:90,1] + 20.072;
   1:  PR[GP1:91,2] = PR[GP1:90,2] + 31.789;
   1:L PR[91] 10mm/sec CNT100;
   1:  PR[GP1:91,1] = PR[GP1:90,1] + 18.409;
   1:  PR[GP1:91,2] = PR[GP1:90,2] + 31.309;
   1:L PR[91] 10mm/sec CNT100;
   1:  PR[GP1:91,1] = PR[GP1:90,1] + 16.069;
   1:  PR[GP1:91,2] = PR[GP1:90,2] + 29.983;
   1:L PR[91] 10mm/sec CNT100;
   1:  PR[GP1:91,1] = PR[GP1:90,1] + 10.473;
   1:  PR[GP1:91,2] = PR[GP1:90,2] + 25.771;
   1:L PR[91] 10mm/sec CNT100;
   1:  PR[GP1:91,1] = PR[GP1:90,1] + 7.432;
   1:  PR[GP1:91,2] = PR[GP1:90,2] + 23.031;
   1:L PR[91] 10mm/sec CNT100;
   1:  PR[GP1:91,1] = PR[GP1:90,1] + 5.247;
   1:  PR[GP1:91,2] = PR[GP1:90,2] + 19.549;
   1:L PR[91] 10mm/sec CNT100;
   1:  PR[GP1:91,1] = PR[GP1:90,1] + 2.029;
   1:  PR[GP1:91,2] = PR[GP1:90,2] + 15.066;
   1:L PR[91] 10mm/sec CNT100;
   1:  PR[GP1:91,1] = PR[GP1:90,1] + -2.576;
   1:L PR[91] 10mm/sec CNT100;
   1:  PR[GP1:91,1] = PR[GP1:90,1] + -4.443;
   1:  PR[GP1:91,2] = PR[GP1:90,2] + 18.006;
   1:L PR[91] 10mm/sec CNT100;
   1:  PR[GP1:91,1] = PR[GP1:90,1] + -7.920;
   1:  PR[GP1:91,2] = PR[GP1:90,2] + 23.001;
   1:L PR[91] 10mm/sec CNT100;
   1:  PR[GP1:91,1] = PR[GP1:90,1] + -10.987;
   1:  PR[GP1:91,2] = PR[GP1:90,2] + 25.765;
   1:L PR[91] 10mm/sec CNT100;
   1:  PR[GP1:91,1] = PR[GP1:90,1] + -16.586;
   1:  PR[GP1:91,2] = PR[GP1:90,2] + 29.971;
   1:L PR[91] 10mm/sec CNT100;
   1:  PR[GP1:91,1] = PR[GP1:90,1] + -18.949;
   1:  PR[GP1:91,2] = PR[GP1:90,2] + 31.314;
   1:L PR[91] 10mm/sec CNT100;
   1:  PR[GP1:91,1] = PR[GP1:90,1] + -30.352;
   1:  PR[GP1:91,2] = PR[GP1:90,2] + 34.913;
   1:L PR[91] 10mm/sec CNT100;
   1:  PR[GP1:91,1] = PR[GP1:90,1] + -42.474;
   1:  PR[GP1:91,2] = PR[GP1:90,2] + 34.813;
   1:L PR[91] 10mm/sec CNT100;
   1:  PR[GP1:91,1] = PR[GP1:90,1] + -45.934;
   1:  PR[GP1:91,2] = PR[GP1:90,2] + 33.714;
   1:L PR[91] 10mm/sec CNT100;
   1:  PR[GP1:91,1] = PR[GP1:90,1] + -54.055;
   1:  PR[GP1:91,2] = PR[GP1:90,2] + 30.773;
   1:L PR[91] 10mm/sec CNT100;
   1:  PR[GP1:91,1] = PR[GP1:90,1] + -59.161;
   1:  PR[GP1:91,2] = PR[GP1:90,2] + 26.808;
   1:L PR[91] 10mm/sec CNT100;
   1:  PR[GP1:91,1] = PR[GP1:90,1] + -63.711;
   1:  PR[GP1:91,2] = PR[GP1:90,2] + 23.056;
   1:L PR[91] 10mm/sec CNT100;
   1:  PR[GP1:91,1] = PR[GP1:90,1] + -67.980;
   1:  PR[GP1:91,2] = PR[GP1:90,2] + 16.084;
   1:L PR[91] 10mm/sec CNT100;
   1:  PR[GP1:91,1] = PR[GP1:90,1] + -70.120;
   1:  PR[GP1:91,2] = PR[GP1:90,2] + 12.435;
   1:L PR[91] 10mm/sec CNT100;
   1:  PR[GP1:91,1] = PR[GP1:90,1] + -71.757;
   1:  PR[GP1:91,2] = PR[GP1:90,2] + 3.678;
   1:L PR[91] 10mm/sec CNT100;
   1:  PR[GP1:91,1] = PR[GP1:90,1] + -71.947;
   1:  PR[GP1:91,2] = PR[GP1:90,2] + 2.795;
   1:L PR[91] 10mm/sec CNT100;
   1:  PR[GP1:91,1] = PR[GP1:90,1] + -72.398;
   1:  PR[GP1:91,2] = PR[GP1:90,2] + 0.282;
   1:L PR[91] 10mm/sec CNT100;
   1:  PR[GP1:91,1] = PR[GP1:90,1] + -70.740;
   1:  PR[GP1:91,2] = PR[GP1:90,2] + -8.405;
   1:L PR[91] 10mm/sec CNT100;
   1:  PR[GP1:91,1] = PR[GP1:90,1] + -70.119;
   1:  PR[GP1:91,2] = PR[GP1:90,2] + -11.880;
   1:L PR[91] 10mm/sec CNT100;
   1:  PR[GP1:91,1] = PR[GP1:90,1] + -67.980;
   1:  PR[GP1:91,2] = PR[GP1:90,2] + -15.525;
   1:L PR[91] 10mm/sec CNT100;
   1:  PR[GP1:91,1] = PR[GP1:90,1] + -63.711;
   1:  PR[GP1:91,2] = PR[GP1:90,2] + -22.498;
   1:L PR[91] 10mm/sec CNT100;
   1:  PR[GP1:91,1] = PR[GP1:90,1] + -59.161;
   1:  PR[GP1:91,2] = PR[GP1:90,2] + -26.250;
   1:L PR[91] 10mm/sec CNT100;
   1:  PR[GP1:91,1] = PR[GP1:90,1] + -54.055;
   1:  PR[GP1:91,2] = PR[GP1:90,2] + -30.215;
   1:L PR[91] 10mm/sec CNT100;
   1:  PR[GP1:91,1] = PR[GP1:90,1] + -45.934;
   1:  PR[GP1:91,2] = PR[GP1:90,2] + -33.156;
   1:L PR[91] 10mm/sec CNT100;
   1:  PR[GP1:91,1] = PR[GP1:90,1] + -42.474;
   1:  PR[GP1:91,2] = PR[GP1:90,2] + -34.255;
   1:L PR[91] 10mm/sec CNT100;
   1:  PR[GP1:91,1] = PR[GP1:90,1] + -30.353;
   1:  PR[GP1:91,2] = PR[GP1:90,2] + -34.355;
   1:L PR[91] 10mm/sec CNT100;
   1:  PR[GP1:91,1] = PR[GP1:90,1] + -20.602;
   1:  PR[GP1:91,2] = PR[GP1:90,2] + -31.231;
   1:L PR[91] 10mm/sec CNT100;
   1:  PR[GP1:91,1] = PR[GP1:90,1] + -18.942;
   1:  PR[GP1:91,2] = PR[GP1:90,2] + -30.752;
   1:L PR[91] 10mm/sec CNT100;
   1:  PR[GP1:91,1] = PR[GP1:90,1] + -16.586;
   1:  PR[GP1:91,2] = PR[GP1:90,2] + -29.413;
   1:L PR[91] 10mm/sec CNT100;
   1:  PR[GP1:91,1] = PR[GP1:90,1] + -10.987;
   1:  PR[GP1:91,2] = PR[GP1:90,2] + -25.207;
   1:L PR[91] 10mm/sec CNT100;
   1:  PR[GP1:91,1] = PR[GP1:90,1] + -7.931;
   1:  PR[GP1:91,2] = PR[GP1:90,2] + -22.452;
   1:L PR[91] 10mm/sec CNT100;
   1:  PR[GP1:91,1] = PR[GP1:90,1] + -5.750;
   1:  PR[GP1:91,2] = PR[GP1:90,2] + -18.972;
   1:L PR[91] 10mm/sec CNT100;
   1:  PR[GP1:91,1] = PR[GP1:90,1] + -2.555;
   1:  PR[GP1:91,2] = PR[GP1:90,2] + -14.507;
   1:L PR[91] 10mm/sec CNT100;
   1:  PR[GP1:91,1] = PR[GP1:90,1] + 2.051;
   1:  PR[GP1:91,2] = PR[GP1:90,2] + -14.508;
   1:L PR[91] 10mm/sec CNT100;
   1:  PR[GP1:91,1] = PR[GP1:90,1] + 3.148;
   1:  PR[GP1:91,2] = PR[GP1:90,2] + -16.727;
   1:  PR[GP1:91,3] = PR[GP1:90,3] + 35.685;
   1:L PR[91] 10mm/sec CNT100;
   1:  PR[GP1:91,1] = PR[GP1:90,1] + 7.151;
   1:  PR[GP1:91,2] = PR[GP1:90,2] + -22.462;
   1:L PR[91] 10mm/sec CNT100;
   1:  PR[GP1:91,1] = PR[GP1:90,1] + 10.644;
   1:  PR[GP1:91,2] = PR[GP1:90,2] + -25.609;
   1:L PR[91] 10mm/sec CNT100;
   1:  PR[GP1:91,1] = PR[GP1:90,1] + 15.427;
   1:  PR[GP1:91,2] = PR[GP1:90,2] + -29.209;
   1:L PR[91] 10mm/sec CNT100;
   1:  PR[GP1:91,1] = PR[GP1:90,1] + 18.388;
   1:  PR[GP1:91,2] = PR[GP1:90,2] + -30.887;
   1:L PR[91] 10mm/sec CNT100;
   1:  PR[GP1:91,1] = PR[GP1:90,1] + 28.617;
   1:  PR[GP1:91,2] = PR[GP1:90,2] + -34.117;
   1:L PR[91] 10mm/sec CNT100;
   1:  PR[GP1:91,1] = PR[GP1:90,1] + 29.505;
   1:  PR[GP1:91,2] = PR[GP1:90,2] + -34.381;
   1:L PR[91] 10mm/sec CNT100;
   1:  PR[GP1:91,1] = PR[GP1:90,1] + 30.004;
   1:  PR[GP1:91,2] = PR[GP1:90,2] + -34.424;
   1:L PR[91] 10mm/sec CNT100;
   1:  PR[GP1:91,1] = PR[GP1:90,1] + 33.129;
   1:  PR[GP1:91,2] = PR[GP1:90,2] + -34.333;
   1:L PR[91] 10mm/sec CNT100;
   1:  PR[GP1:91,1] = PR[GP1:90,1] + 41.923;
   1:  PR[GP1:91,2] = PR[GP1:90,2] + -34.263;
   1:L PR[91] 10mm/sec CNT100;
   1:  PR[GP1:91,1] = PR[GP1:90,1] + 44.482;
   1:  PR[GP1:91,2] = PR[GP1:90,2] + -33.451;
   1:L PR[91] 10mm/sec CNT100;
   1:  PR[GP1:91,1] = PR[GP1:90,1] + 53.470;
   1:  PR[GP1:91,2] = PR[GP1:90,2] + -30.199;
   1:L PR[91] 10mm/sec CNT100;
   1:  PR[GP1:91,1] = PR[GP1:90,1] + 57.908;
   1:  PR[GP1:91,2] = PR[GP1:90,2] + -26.751;
   1:L PR[91] 10mm/sec CNT100;
   1:  PR[GP1:91,1] = PR[GP1:90,1] + 63.095;
   1:  PR[GP1:91,2] = PR[GP1:90,2] + -22.469;
   1:L PR[91] 10mm/sec CNT100;
   1:  PR[GP1:91,1] = PR[GP1:90,1] + 66.968;
   1:  PR[GP1:91,2] = PR[GP1:90,2] + -16.153;
   1:L PR[91] 10mm/sec CNT100;
   1:  PR[GP1:91,1] = PR[GP1:90,1] + 69.485;
   1:  PR[GP1:91,2] = PR[GP1:90,2] + -11.876;
   1:L PR[91] 10mm/sec CNT100;
   1:  PR[GP1:91,1] = PR[GP1:90,1] + 70.993;
   1:  PR[GP1:91,2] = PR[GP1:90,2] + -3.797;
   1:L PR[91] 10mm/sec CNT100;
   1:  PR[GP1:91,1] = PR[GP1:90,1] + 71.169;
   1:  PR[GP1:91,2] = PR[GP1:90,2] + -2.980;
   1:L PR[91] 10mm/sec CNT100;
   1:  PR[GP1:91,1] = PR[GP1:90,1] + 71.752;
   1:  PR[GP1:91,2] = PR[GP1:90,2] + 0.276;
   1:L PR[91] 10mm/sec CNT100;
   1:  PR[GP1:91,1] = PR[GP1:90,1] + 70.214;
   1:  PR[GP1:91,2] = PR[GP1:90,2] + 8.343;
   1:L PR[91] 10mm/sec CNT100;
   1:  PR[GP1:91,1] = PR[GP1:90,1] + 69.484;
   1:  PR[GP1:91,2] = PR[GP1:90,2] + 12.437;
   1:L PR[91] 10mm/sec CNT100;
   1:  PR[GP1:91,1] = PR[GP1:90,1] + 66.968;
   1:  PR[GP1:91,2] = PR[GP1:90,2] + 16.711;
   1:L PR[91] 10mm/sec CNT100;
   1:  PR[GP1:91,1] = PR[GP1:90,1] + 63.095;
   1:  PR[GP1:91,2] = PR[GP1:90,2] + 23.027;
   1:L PR[91] 10mm/sec CNT100;
   1:  PR[GP1:91,1] = PR[GP1:90,1] + 57.908;
   1:  PR[GP1:91,2] = PR[GP1:90,2] + 27.309;
   1:L PR[91] 10mm/sec CNT100;
   1:  PR[GP1:91,1] = PR[GP1:90,1] + 53.470;
   1:  PR[GP1:91,2] = PR[GP1:90,2] + 30.757;
   1:L PR[91] 10mm/sec CNT100;
   1:  PR[GP1:91,1] = PR[GP1:90,1] + 44.482;
   1:  PR[GP1:91,2] = PR[GP1:90,2] + 34.009;
   1:L PR[91] 10mm/sec CNT100;
   1:  PR[GP1:91,1] = PR[GP1:90,1] + 41.923;
   1:  PR[GP1:91,2] = PR[GP1:90,2] + 34.821;
   1:L PR[91] 10mm/sec CNT100;
   1:  PR[GP1:91,1] = PR[GP1:90,1] + 33.129;
   1:  PR[GP1:91,2] = PR[GP1:90,2] + 34.891;
   1:L PR[91] 10mm/sec CNT100;
   1:  PR[GP1:91,1] = PR[GP1:90,1] + 30.004;
   1:  PR[GP1:91,2] = PR[GP1:90,2] + 34.982;
   1:L PR[91] 10mm/sec CNT100;
   1:  PR[GP1:91,1] = PR[GP1:90,1] + 29.511;
   1:  PR[GP1:91,2] = PR[GP1:90,2] + 34.940;
   1:L PR[91] 10mm/sec CNT100;
   1:  PR[GP1:91,1] = PR[GP1:90,1] + 20.479;
   1:  PR[GP1:91,2] = PR[GP1:90,2] + 32.046;
   1:L PR[91] 10mm/sec CNT100;
   1:  PR[GP1:91,1] = PR[GP1:90,1] + 18.382;
   1:  PR[GP1:91,2] = PR[GP1:90,2] + 31.441;
   1:L PR[91] 10mm/sec CNT100;
   1:  PR[GP1:91,1] = PR[GP1:90,1] + 15.427;
   1:  PR[GP1:91,2] = PR[GP1:90,2] + 29.767;
   1:L PR[91] 10mm/sec CNT100;
   1:  PR[GP1:91,1] = PR[GP1:90,1] + 10.644;
   1:  PR[GP1:91,2] = PR[GP1:90,2] + 26.167;
   1:L PR[91] 10mm/sec CNT100;
   1:  PR[GP1:91,1] = PR[GP1:90,1] + 7.162;
   1:  PR[GP1:91,2] = PR[GP1:90,2] + 23.030;
   1:L PR[91] 10mm/sec CNT100;
   1:  PR[GP1:91,1] = PR[GP1:90,1] + 5.472;
   1:  PR[GP1:91,2] = PR[GP1:90,2] + 20.336;
   1:L PR[91] 10mm/sec CNT100;
   1:  PR[GP1:91,1] = PR[GP1:90,1] + 1.922;
   1:  PR[GP1:91,2] = PR[GP1:90,2] + 15.391;
   1:L PR[91] 10mm/sec CNT100;
   1:  PR[GP1:91,1] = PR[GP1:90,1] + -2.468;
   1:L PR[91] 10mm/sec CNT100;
   1:  PR[GP1:91,1] = PR[GP1:90,1] + -3.672;
   1:  PR[GP1:91,2] = PR[GP1:90,2] + 17.286;
   1:L PR[91] 10mm/sec CNT100;
   1:  PR[GP1:91,1] = PR[GP1:90,1] + -7.645;
   1:  PR[GP1:91,2] = PR[GP1:90,2] + 22.994;
   1:L PR[91] 10mm/sec CNT100;
   1:  PR[GP1:91,1] = PR[GP1:90,1] + -11.155;
   1:  PR[GP1:91,2] = PR[GP1:90,2] + 26.157;
   1:L PR[91] 10mm/sec CNT100;
   1:  PR[GP1:91,1] = PR[GP1:90,1] + -15.939;
   1:  PR[GP1:91,2] = PR[GP1:90,2] + 29.752;
   1:L PR[91] 10mm/sec CNT100;
   1:  PR[GP1:91,1] = PR[GP1:90,1] + -18.921;
   1:  PR[GP1:91,2] = PR[GP1:90,2] + 31.447;
   1:L PR[91] 10mm/sec CNT100;
   1:  PR[GP1:91,1] = PR[GP1:90,1] + -29.151;
   1:  PR[GP1:91,2] = PR[GP1:90,2] + 34.677;
   1:L PR[91] 10mm/sec CNT100;
   1:  PR[GP1:91,1] = PR[GP1:90,1] + -30.037;
   1:  PR[GP1:91,2] = PR[GP1:90,2] + 34.940;
   1:L PR[91] 10mm/sec CNT100;
   1:  PR[GP1:91,1] = PR[GP1:90,1] + -30.536;
   1:  PR[GP1:91,2] = PR[GP1:90,2] + 34.983;
   1:L PR[91] 10mm/sec CNT100;
   1:  PR[GP1:91,1] = PR[GP1:90,1] + -33.655;
   1:  PR[GP1:91,2] = PR[GP1:90,2] + 34.891;
   1:L PR[91] 10mm/sec CNT100;
   1:  PR[GP1:91,1] = PR[GP1:90,1] + -42.455;
   1:  PR[GP1:91,2] = PR[GP1:90,2] + 34.820;
   1:L PR[91] 10mm/sec CNT100;
   1:  PR[GP1:91,1] = PR[GP1:90,1] + -45.014;
   1:  PR[GP1:91,2] = PR[GP1:90,2] + 34.007;
   1:L PR[91] 10mm/sec CNT100;
   1:  PR[GP1:91,1] = PR[GP1:90,1] + -54.001;
   1:  PR[GP1:91,2] = PR[GP1:90,2] + 30.753;
   1:L PR[91] 10mm/sec CNT100;
   1:  PR[GP1:91,1] = PR[GP1:90,1] + -58.439;
   1:  PR[GP1:91,2] = PR[GP1:90,2] + 27.306;
   1:L PR[91] 10mm/sec CNT100;
   1:  PR[GP1:91,1] = PR[GP1:90,1] + -63.624;
   1:  PR[GP1:91,2] = PR[GP1:90,2] + 23.030;
   1:L PR[91] 10mm/sec CNT100;
   1:  PR[GP1:91,1] = PR[GP1:90,1] + -67.496;
   1:  PR[GP1:91,2] = PR[GP1:90,2] + 16.707;
   1:L PR[91] 10mm/sec CNT100;
   1:  PR[GP1:91,1] = PR[GP1:90,1] + -70.012;
   1:  PR[GP1:91,2] = PR[GP1:90,2] + 12.419;
   1:L PR[91] 10mm/sec CNT100;
   1:  PR[GP1:91,1] = PR[GP1:90,1] + -71.520;
   1:  PR[GP1:91,2] = PR[GP1:90,2] + 4.347;
   1:L PR[91] 10mm/sec CNT100;
   1:  PR[GP1:91,1] = PR[GP1:90,1] + -71.696;
   1:  PR[GP1:91,2] = PR[GP1:90,2] + 3.532;
   1:L PR[91] 10mm/sec CNT100;
   1:  PR[GP1:91,1] = PR[GP1:90,1] + -72.278;
   1:  PR[GP1:91,2] = PR[GP1:90,2] + 0.282;
   1:L PR[91] 10mm/sec CNT100;
   1:  PR[GP1:91,1] = PR[GP1:90,1] + -70.741;
   1:  PR[GP1:91,2] = PR[GP1:90,2] + -7.776;
   1:L PR[91] 10mm/sec CNT100;
   1:  PR[GP1:91,1] = PR[GP1:90,1] + -70.011;
   1:  PR[GP1:91,2] = PR[GP1:90,2] + -11.863;
   1:L PR[91] 10mm/sec CNT100;
   1:  PR[GP1:91,1] = PR[GP1:90,1] + -67.496;
   1:  PR[GP1:91,2] = PR[GP1:90,2] + -16.149;
   1:L PR[91] 10mm/sec CNT100;
   1:  PR[GP1:91,1] = PR[GP1:90,1] + -63.624;
   1:  PR[GP1:91,2] = PR[GP1:90,2] + -22.472;
   1:L PR[91] 10mm/sec CNT100;
   1:  PR[GP1:91,1] = PR[GP1:90,1] + -58.439;
   1:  PR[GP1:91,2] = PR[GP1:90,2] + -26.748;
   1:L PR[91] 10mm/sec CNT100;
   1:  PR[GP1:91,1] = PR[GP1:90,1] + -54.001;
   1:  PR[GP1:91,2] = PR[GP1:90,2] + -30.195;
   1:L PR[91] 10mm/sec CNT100;
   1:  PR[GP1:91,1] = PR[GP1:90,1] + -45.014;
   1:  PR[GP1:91,2] = PR[GP1:90,2] + -33.449;
   1:L PR[91] 10mm/sec CNT100;
   1:  PR[GP1:91,1] = PR[GP1:90,1] + -42.455;
   1:  PR[GP1:91,2] = PR[GP1:90,2] + -34.262;
   1:L PR[91] 10mm/sec CNT100;
   1:  PR[GP1:91,1] = PR[GP1:90,1] + -33.655;
   1:  PR[GP1:91,2] = PR[GP1:90,2] + -34.333;
   1:L PR[91] 10mm/sec CNT100;
   1:  PR[GP1:91,1] = PR[GP1:90,1] + -30.536;
   1:  PR[GP1:91,2] = PR[GP1:90,2] + -34.425;
   1:L PR[91] 10mm/sec CNT100;
   1:  PR[GP1:91,1] = PR[GP1:90,1] + -30.043;
   1:  PR[GP1:91,2] = PR[GP1:90,2] + -34.382;
   1:L PR[91] 10mm/sec CNT100;
   1:  PR[GP1:91,1] = PR[GP1:90,1] + -21.009;
   1:  PR[GP1:91,2] = PR[GP1:90,2] + -31.488;
   1:L PR[91] 10mm/sec CNT100;
   1:  PR[GP1:91,1] = PR[GP1:90,1] + -18.915;
   1:  PR[GP1:91,2] = PR[GP1:90,2] + -30.885;
   1:L PR[91] 10mm/sec CNT100;
   1:  PR[GP1:91,1] = PR[GP1:90,1] + -15.939;
   1:  PR[GP1:91,2] = PR[GP1:90,2] + -29.194;
   1:L PR[91] 10mm/sec CNT100;
   1:  PR[GP1:91,1] = PR[GP1:90,1] + -11.155;
   1:  PR[GP1:91,2] = PR[GP1:90,2] + -25.599;
   1:L PR[91] 10mm/sec CNT100;
   1:  PR[GP1:91,1] = PR[GP1:90,1] + -7.656;
   1:  PR[GP1:91,2] = PR[GP1:90,2] + -22.446;
   1:L PR[91] 10mm/sec CNT100;
   1:  PR[GP1:91,1] = PR[GP1:90,1] + -5.971;
   1:  PR[GP1:91,2] = PR[GP1:90,2] + -19.757;
   1:L PR[91] 10mm/sec CNT100;
   1:  PR[GP1:91,1] = PR[GP1:90,1] + -2.447;
   1:  PR[GP1:91,2] = PR[GP1:90,2] + -14.832;
   1:L PR[91] 10mm/sec CNT100;
   1:  PR[GP1:91,1] = PR[GP1:90,1] + 1.944;
   1:L PR[91] 10mm/sec CNT100;
   1:  PR[GP1:91,1] = PR[GP1:90,1] + 2.378;
   1:  PR[GP1:91,2] = PR[GP1:90,2] + -16.009;
   1:  PR[GP1:91,3] = PR[GP1:90,3] + 36.295;
   1:L PR[91] 10mm/sec CNT100;
   1:  PR[GP1:91,1] = PR[GP1:90,1] + 6.881;
   1:  PR[GP1:91,2] = PR[GP1:90,2] + -22.460;
   1:L PR[91] 10mm/sec CNT100;
   1:  PR[GP1:91,1] = PR[GP1:90,1] + 10.814;
   1:  PR[GP1:91,2] = PR[GP1:90,2] + -26.004;
   1:L PR[91] 10mm/sec CNT100;
   1:  PR[GP1:91,1] = PR[GP1:90,1] + 14.785;
   1:  PR[GP1:91,2] = PR[GP1:90,2] + -28.993;
   1:L PR[91] 10mm/sec CNT100;
   1:  PR[GP1:91,1] = PR[GP1:90,1] + 18.361;
   1:  PR[GP1:91,2] = PR[GP1:90,2] + -31.019;
   1:L PR[91] 10mm/sec CNT100;
   1:  PR[GP1:91,1] = PR[GP1:90,1] + 27.435;
   1:  PR[GP1:91,2] = PR[GP1:90,2] + -33.884;
   1:L PR[91] 10mm/sec CNT100;
   1:  PR[GP1:91,1] = PR[GP1:90,1] + 29.168;
   1:  PR[GP1:91,2] = PR[GP1:90,2] + -34.400;
   1:L PR[91] 10mm/sec CNT100;
   1:  PR[GP1:91,1] = PR[GP1:90,1] + 30.195;
   1:  PR[GP1:91,2] = PR[GP1:90,2] + -34.489;
   1:L PR[91] 10mm/sec CNT100;
   1:  PR[GP1:91,1] = PR[GP1:90,1] + 36.121;
   1:  PR[GP1:91,2] = PR[GP1:90,2] + -34.316;
   1:L PR[91] 10mm/sec CNT100;
   1:  PR[GP1:91,1] = PR[GP1:90,1] + 41.905;
   1:  PR[GP1:91,2] = PR[GP1:90,2] + -34.270;
   1:L PR[91] 10mm/sec CNT100;
   1:  PR[GP1:91,1] = PR[GP1:90,1] + 43.563;
   1:  PR[GP1:91,2] = PR[GP1:90,2] + -33.743;
   1:L PR[91] 10mm/sec CNT100;
   1:  PR[GP1:91,1] = PR[GP1:90,1] + 53.416;
   1:  PR[GP1:91,2] = PR[GP1:90,2] + -30.179;
   1:L PR[91] 10mm/sec CNT100;
   1:  PR[GP1:91,1] = PR[GP1:90,1] + 57.186;
   1:  PR[GP1:91,2] = PR[GP1:90,2] + -27.250;
   1:L PR[91] 10mm/sec CNT100;
   1:  PR[GP1:91,1] = PR[GP1:90,1] + 63.008;
   1:  PR[GP1:91,2] = PR[GP1:90,2] + -22.443;
   1:L PR[91] 10mm/sec CNT100;
   1:  PR[GP1:91,1] = PR[GP1:90,1] + 66.484;
   1:  PR[GP1:91,2] = PR[GP1:90,2] + -16.775;
   1:L PR[91] 10mm/sec CNT100;
   1:  PR[GP1:91,1] = PR[GP1:90,1] + 69.376;
   1:  PR[GP1:91,2] = PR[GP1:90,2] + -11.860;
   1:L PR[91] 10mm/sec CNT100;
   1:  PR[GP1:91,1] = PR[GP1:90,1] + 70.757;
   1:  PR[GP1:91,2] = PR[GP1:90,2] + -4.466;
   1:L PR[91] 10mm/sec CNT100;
   1:  PR[GP1:91,1] = PR[GP1:90,1] + 70.918;
   1:  PR[GP1:91,2] = PR[GP1:90,2] + -3.719;
   1:L PR[91] 10mm/sec CNT100;
   1:  PR[GP1:91,1] = PR[GP1:90,1] + 71.633;
   1:  PR[GP1:91,2] = PR[GP1:90,2] + 0.276;
   1:L PR[91] 10mm/sec CNT100;
   1:  PR[GP1:91,1] = PR[GP1:90,1] + 70.215;
   1:  PR[GP1:91,2] = PR[GP1:90,2] + 7.714;
   1:L PR[91] 10mm/sec CNT100;
   1:  PR[GP1:91,1] = PR[GP1:90,1] + 69.375;
   1:  PR[GP1:91,2] = PR[GP1:90,2] + 12.420;
   1:L PR[91] 10mm/sec CNT100;
   1:  PR[GP1:91,1] = PR[GP1:90,1] + 66.484;
   1:  PR[GP1:91,2] = PR[GP1:90,2] + 17.333;
   1:L PR[91] 10mm/sec CNT100;
   1:  PR[GP1:91,1] = PR[GP1:90,1] + 63.008;
   1:  PR[GP1:91,2] = PR[GP1:90,2] + 23.001;
   1:L PR[91] 10mm/sec CNT100;
   1:  PR[GP1:91,1] = PR[GP1:90,1] + 57.187;
   1:  PR[GP1:91,2] = PR[GP1:90,2] + 27.808;
   1:L PR[91] 10mm/sec CNT100;
   1:  PR[GP1:91,1] = PR[GP1:90,1] + 53.416;
   1:  PR[GP1:91,2] = PR[GP1:90,2] + 30.737;
   1:L PR[91] 10mm/sec CNT100;
   1:  PR[GP1:91,1] = PR[GP1:90,1] + 43.563;
   1:  PR[GP1:91,2] = PR[GP1:90,2] + 34.301;
   1:L PR[91] 10mm/sec CNT100;
   1:  PR[GP1:91,1] = PR[GP1:90,1] + 41.905;
   1:  PR[GP1:91,2] = PR[GP1:90,2] + 34.828;
   1:L PR[91] 10mm/sec CNT100;
   1:  PR[GP1:91,1] = PR[GP1:90,1] + 36.121;
   1:  PR[GP1:91,2] = PR[GP1:90,2] + 34.874;
   1:L PR[91] 10mm/sec CNT100;
   1:  PR[GP1:91,1] = PR[GP1:90,1] + 30.195;
   1:  PR[GP1:91,2] = PR[GP1:90,2] + 35.047;
   1:L PR[91] 10mm/sec CNT100;
   1:  PR[GP1:91,1] = PR[GP1:90,1] + 29.175;
   1:  PR[GP1:91,2] = PR[GP1:90,2] + 34.959;
   1:L PR[91] 10mm/sec CNT100;
   1:  PR[GP1:91,1] = PR[GP1:90,1] + 20.887;
   1:  PR[GP1:91,2] = PR[GP1:90,2] + 32.304;
   1:L PR[91] 10mm/sec CNT100;
   1:  PR[GP1:91,1] = PR[GP1:90,1] + 18.354;
   1:  PR[GP1:91,2] = PR[GP1:90,2] + 31.574;
   1:L PR[91] 10mm/sec CNT100;
   1:  PR[GP1:91,1] = PR[GP1:90,1] + 14.785;
   1:  PR[GP1:91,2] = PR[GP1:90,2] + 29.551;
   1:L PR[91] 10mm/sec CNT100;
   1:  PR[GP1:91,1] = PR[GP1:90,1] + 10.814;
   1:  PR[GP1:91,2] = PR[GP1:90,2] + 26.562;
   1:L PR[91] 10mm/sec CNT100;
   1:  PR[GP1:91,1] = PR[GP1:90,1] + 6.892;
   1:  PR[GP1:91,2] = PR[GP1:90,2] + 23.029;
   1:L PR[91] 10mm/sec CNT100;
   1:  PR[GP1:91,1] = PR[GP1:90,1] + 5.696;
   1:  PR[GP1:91,2] = PR[GP1:90,2] + 21.123;
   1:L PR[91] 10mm/sec CNT100;
   1:  PR[GP1:91,1] = PR[GP1:90,1] + 1.816;
   1:  PR[GP1:91,2] = PR[GP1:90,2] + 15.715;
   1:L PR[91] 10mm/sec CNT100;
   1:  PR[GP1:91,1] = PR[GP1:90,1] + -2.360;
   1:L PR[91] 10mm/sec CNT100;
   1:  PR[GP1:91,1] = PR[GP1:90,1] + -2.901;
   1:  PR[GP1:91,2] = PR[GP1:90,2] + 16.566;
   1:L PR[91] 10mm/sec CNT100;
   1:  PR[GP1:91,1] = PR[GP1:90,1] + -7.371;
   1:  PR[GP1:91,2] = PR[GP1:90,2] + 22.988;
   1:L PR[91] 10mm/sec CNT100;
   1:  PR[GP1:91,1] = PR[GP1:90,1] + -11.323;
   1:  PR[GP1:91,2] = PR[GP1:90,2] + 26.550;
   1:L PR[91] 10mm/sec CNT100;
   1:  PR[GP1:91,1] = PR[GP1:90,1] + -15.293;
   1:  PR[GP1:91,2] = PR[GP1:90,2] + 29.533;
   1:L PR[91] 10mm/sec CNT100;
   1:  PR[GP1:91,1] = PR[GP1:90,1] + -18.894;
   1:  PR[GP1:91,2] = PR[GP1:90,2] + 31.579;
   1:L PR[91] 10mm/sec CNT100;
   1:  PR[GP1:91,1] = PR[GP1:90,1] + -27.970;
   1:  PR[GP1:91,2] = PR[GP1:90,2] + 34.445;
   1:L PR[91] 10mm/sec CNT100;
   1:  PR[GP1:91,1] = PR[GP1:90,1] + -29.699;
   1:  PR[GP1:91,2] = PR[GP1:90,2] + 34.959;
   1:L PR[91] 10mm/sec CNT100;
   1:  PR[GP1:91,1] = PR[GP1:90,1] + -30.728;
   1:  PR[GP1:91,2] = PR[GP1:90,2] + 35.047;
   1:L PR[91] 10mm/sec CNT100;
   1:  PR[GP1:91,1] = PR[GP1:90,1] + -36.647;
   1:  PR[GP1:91,2] = PR[GP1:90,2] + 34.874;
   1:L PR[91] 10mm/sec CNT100;
   1:  PR[GP1:91,1] = PR[GP1:90,1] + -42.436;
   1:  PR[GP1:91,2] = PR[GP1:90,2] + 34.827;
   1:L PR[91] 10mm/sec CNT100;
   1:  PR[GP1:91,1] = PR[GP1:90,1] + -44.095;
   1:  PR[GP1:91,2] = PR[GP1:90,2] + 34.300;
   1:L PR[91] 10mm/sec CNT100;
   1:  PR[GP1:91,1] = PR[GP1:90,1] + -53.946;
   1:  PR[GP1:91,2] = PR[GP1:90,2] + 30.732;
   1:L PR[91] 10mm/sec CNT100;
   1:  PR[GP1:91,1] = PR[GP1:90,1] + -57.717;
   1:  PR[GP1:91,2] = PR[GP1:90,2] + 27.804;
   1:L PR[91] 10mm/sec CNT100;
   1:  PR[GP1:91,1] = PR[GP1:90,1] + -63.537;
   1:  PR[GP1:91,2] = PR[GP1:90,2] + 23.004;
   1:L PR[91] 10mm/sec CNT100;
   1:  PR[GP1:91,1] = PR[GP1:90,1] + -67.012;
   1:  PR[GP1:91,2] = PR[GP1:90,2] + 17.330;
   1:L PR[91] 10mm/sec CNT100;
   1:  PR[GP1:91,1] = PR[GP1:90,1] + -69.903;
   1:  PR[GP1:91,2] = PR[GP1:90,2] + 12.402;
   1:L PR[91] 10mm/sec CNT100;
   1:  PR[GP1:91,1] = PR[GP1:90,1] + -71.283;
   1:  PR[GP1:91,2] = PR[GP1:90,2] + 5.016;
   1:L PR[91] 10mm/sec CNT100;
   1:  PR[GP1:91,1] = PR[GP1:90,1] + -71.444;
   1:  PR[GP1:91,2] = PR[GP1:90,2] + 4.269;
   1:L PR[91] 10mm/sec CNT100;
   1:  PR[GP1:91,1] = PR[GP1:90,1] + -72.159;
   1:  PR[GP1:91,2] = PR[GP1:90,2] + 0.282;
   1:L PR[91] 10mm/sec CNT100;
   1:  PR[GP1:91,1] = PR[GP1:90,1] + -70.741;
   1:  PR[GP1:91,2] = PR[GP1:90,2] + -7.148;
   1:L PR[91] 10mm/sec CNT100;
   1:  PR[GP1:91,1] = PR[GP1:90,1] + -69.902;
   1:  PR[GP1:91,2] = PR[GP1:90,2] + -11.846;
   1:L PR[91] 10mm/sec CNT100;
   1:  PR[GP1:91,1] = PR[GP1:90,1] + -67.012;
   1:  PR[GP1:91,2] = PR[GP1:90,2] + -16.772;
   1:L PR[91] 10mm/sec CNT100;
   1:  PR[GP1:91,1] = PR[GP1:90,1] + -63.537;
   1:  PR[GP1:91,2] = PR[GP1:90,2] + -22.446;
   1:L PR[91] 10mm/sec CNT100;
   1:  PR[GP1:91,1] = PR[GP1:90,1] + -57.717;
   1:  PR[GP1:91,2] = PR[GP1:90,2] + -27.246;
   1:L PR[91] 10mm/sec CNT100;
   1:  PR[GP1:91,1] = PR[GP1:90,1] + -53.946;
   1:  PR[GP1:91,2] = PR[GP1:90,2] + -30.174;
   1:L PR[91] 10mm/sec CNT100;
   1:  PR[GP1:91,1] = PR[GP1:90,1] + -44.095;
   1:  PR[GP1:91,2] = PR[GP1:90,2] + -33.742;
   1:L PR[91] 10mm/sec CNT100;
   1:  PR[GP1:91,1] = PR[GP1:90,1] + -42.436;
   1:  PR[GP1:91,2] = PR[GP1:90,2] + -34.269;
   1:L PR[91] 10mm/sec CNT100;
   1:  PR[GP1:91,1] = PR[GP1:90,1] + -36.647;
   1:  PR[GP1:91,2] = PR[GP1:90,2] + -34.316;
   1:L PR[91] 10mm/sec CNT100;
   1:  PR[GP1:91,1] = PR[GP1:90,1] + -30.728;
   1:  PR[GP1:91,2] = PR[GP1:90,2] + -34.489;
   1:L PR[91] 10mm/sec CNT100;
   1:  PR[GP1:91,1] = PR[GP1:90,1] + -29.706;
   1:  PR[GP1:91,2] = PR[GP1:90,2] + -34.402;
   1:L PR[91] 10mm/sec CNT100;
   1:  PR[GP1:91,1] = PR[GP1:90,1] + -21.416;
   1:  PR[GP1:91,2] = PR[GP1:90,2] + -31.746;
   1:L PR[91] 10mm/sec CNT100;
   1:  PR[GP1:91,1] = PR[GP1:90,1] + -18.887;
   1:  PR[GP1:91,2] = PR[GP1:90,2] + -31.017;
   1:L PR[91] 10mm/sec CNT100;
   1:  PR[GP1:91,1] = PR[GP1:90,1] + -15.293;
   1:  PR[GP1:91,2] = PR[GP1:90,2] + -28.974;
   1:L PR[91] 10mm/sec CNT100;
   1:  PR[GP1:91,1] = PR[GP1:90,1] + -11.323;
   1:  PR[GP1:91,2] = PR[GP1:90,2] + -25.992;
   1:L PR[91] 10mm/sec CNT100;
   1:  PR[GP1:91,1] = PR[GP1:90,1] + -7.382;
   1:  PR[GP1:91,2] = PR[GP1:90,2] + -22.440;
   1:L PR[91] 10mm/sec CNT100;
   1:  PR[GP1:91,1] = PR[GP1:90,1] + -6.193;
   1:  PR[GP1:91,2] = PR[GP1:90,2] + -20.543;
   1:L PR[91] 10mm/sec CNT100;
   1:  PR[GP1:91,1] = PR[GP1:90,1] + -2.339;
   1:  PR[GP1:91,2] = PR[GP1:90,2] + -15.157;
   1:L PR[91] 10mm/sec CNT100;
   1:  PR[GP1:91,1] = PR[GP1:90,1] + 1.837;
   1:L PR[91] 10mm/sec CNT100;
   1:  PR[GP1:91,1] = PR[GP1:90,1] + 2.923;
   1:  PR[GP1:91,2] = PR[GP1:90,2] + -17.174;
   1:  PR[GP1:91,3] = PR[GP1:90,3] + 36.905;
   1:L PR[91] 10mm/sec CNT100;
   1:  PR[GP1:91,1] = PR[GP1:90,1] + 6.611;
   1:  PR[GP1:91,2] = PR[GP1:90,2] + -22.459;
   1:L PR[91] 10mm/sec CNT100;
   1:  PR[GP1:91,1] = PR[GP1:90,1] + 10.984;
   1:  PR[GP1:91,2] = PR[GP1:90,2] + -26.399;
   1:L PR[91] 10mm/sec CNT100;
   1:  PR[GP1:91,1] = PR[GP1:90,1] + 14.143;
   1:  PR[GP1:91,2] = PR[GP1:90,2] + -28.777;
   1:L PR[91] 10mm/sec CNT100;
   1:  PR[GP1:91,1] = PR[GP1:90,1] + 18.334;
   1:  PR[GP1:91,2] = PR[GP1:90,2] + -31.151;
   1:L PR[91] 10mm/sec CNT100;
   1:  PR[GP1:91,1] = PR[GP1:90,1] + 26.253;
   1:  PR[GP1:91,2] = PR[GP1:90,2] + -33.652;
   1:L PR[91] 10mm/sec CNT100;
   1:  PR[GP1:91,1] = PR[GP1:90,1] + 28.832;
   1:  PR[GP1:91,2] = PR[GP1:90,2] + -34.419;
   1:L PR[91] 10mm/sec CNT100;
   1:  PR[GP1:91,1] = PR[GP1:90,1] + 30.386;
   1:  PR[GP1:91,2] = PR[GP1:90,2] + -34.553;
   1:L PR[91] 10mm/sec CNT100;
   1:  PR[GP1:91,1] = PR[GP1:90,1] + 39.112;
   1:  PR[GP1:91,2] = PR[GP1:90,2] + -34.298;
   1:L PR[91] 10mm/sec CNT100;
   1:  PR[GP1:91,1] = PR[GP1:90,1] + 41.886;
   1:  PR[GP1:91,2] = PR[GP1:90,2] + -34.276;
   1:L PR[91] 10mm/sec CNT100;
   1:  PR[GP1:91,1] = PR[GP1:90,1] + 42.643;
   1:  PR[GP1:91,2] = PR[GP1:90,2] + -34.036;
   1:L PR[91] 10mm/sec CNT100;
   1:  PR[GP1:91,1] = PR[GP1:90,1] + 53.361;
   1:  PR[GP1:91,2] = PR[GP1:90,2] + -30.159;
   1:L PR[91] 10mm/sec CNT100;
   1:  PR[GP1:91,1] = PR[GP1:90,1] + 56.465;
   1:  PR[GP1:91,2] = PR[GP1:90,2] + -27.748;
   1:L PR[91] 10mm/sec CNT100;
   1:  PR[GP1:91,1] = PR[GP1:90,1] + 62.922;
   1:  PR[GP1:91,2] = PR[GP1:90,2] + -22.417;
   1:L PR[91] 10mm/sec CNT100;
   1:  PR[GP1:91,1] = PR[GP1:90,1] + 66.000;
   1:  PR[GP1:91,2] = PR[GP1:90,2] + -17.397;
   1:L PR[91] 10mm/sec CNT100;
   1:  PR[GP1:91,1] = PR[GP1:90,1] + 69.268;
   1:  PR[GP1:91,2] = PR[GP1:90,2] + -11.844;
   1:L PR[91] 10mm/sec CNT100;
   1:  PR[GP1:91,1] = PR[GP1:90,1] + 70.520;
   1:  PR[GP1:91,2] = PR[GP1:90,2] + -5.136;
   1:L PR[91] 10mm/sec CNT100;
   1:  PR[GP1:91,1] = PR[GP1:90,1] + 70.666;
   1:  PR[GP1:91,2] = PR[GP1:90,2] + -4.457;
   1:L PR[91] 10mm/sec CNT100;
   1:  PR[GP1:91,1] = PR[GP1:90,1] + 71.514;
   1:  PR[GP1:91,2] = PR[GP1:90,2] + 0.276;
   1:L PR[91] 10mm/sec CNT100;
   1:  PR[GP1:91,1] = PR[GP1:90,1] + 70.215;
   1:  PR[GP1:91,2] = PR[GP1:90,2] + 7.085;
   1:L PR[91] 10mm/sec CNT100;
   1:  PR[GP1:91,1] = PR[GP1:90,1] + 69.266;
   1:  PR[GP1:91,2] = PR[GP1:90,2] + 12.404;
   1:L PR[91] 10mm/sec CNT100;
   1:  PR[GP1:91,1] = PR[GP1:90,1] + 66.000;
   1:  PR[GP1:91,2] = PR[GP1:90,2] + 17.955;
   1:L PR[91] 10mm/sec CNT100;
   1:  PR[GP1:91,1] = PR[GP1:90,1] + 62.922;
   1:  PR[GP1:91,2] = PR[GP1:90,2] + 22.975;
   1:L PR[91] 10mm/sec CNT100;
   1:  PR[GP1:91,1] = PR[GP1:90,1] + 56.465;
   1:  PR[GP1:91,2] = PR[GP1:90,2] + 28.306;
   1:L PR[91] 10mm/sec CNT100;
   1:  PR[GP1:91,1] = PR[GP1:90,1] + 53.361;
   1:  PR[GP1:91,2] = PR[GP1:90,2] + 30.717;
   1:L PR[91] 10mm/sec CNT100;
   1:  PR[GP1:91,1] = PR[GP1:90,1] + 42.643;
   1:  PR[GP1:91,2] = PR[GP1:90,2] + 34.594;
   1:L PR[91] 10mm/sec CNT100;
   1:  PR[GP1:91,1] = PR[GP1:90,1] + 41.886;
   1:  PR[GP1:91,2] = PR[GP1:90,2] + 34.834;
   1:L PR[91] 10mm/sec CNT100;
   1:  PR[GP1:91,1] = PR[GP1:90,1] + 39.112;
   1:  PR[GP1:91,2] = PR[GP1:90,2] + 34.856;
   1:L PR[91] 10mm/sec CNT100;
   1:  PR[GP1:91,1] = PR[GP1:90,1] + 30.386;
   1:  PR[GP1:91,2] = PR[GP1:90,2] + 35.111;
   1:L PR[91] 10mm/sec CNT100;
   1:  PR[GP1:91,1] = PR[GP1:90,1] + 28.838;
   1:  PR[GP1:91,2] = PR[GP1:90,2] + 34.978;
   1:L PR[91] 10mm/sec CNT100;
   1:  PR[GP1:91,1] = PR[GP1:90,1] + 21.294;
   1:  PR[GP1:91,2] = PR[GP1:90,2] + 32.561;
   1:L PR[91] 10mm/sec CNT100;
   1:  PR[GP1:91,1] = PR[GP1:90,1] + 18.327;
   1:  PR[GP1:91,2] = PR[GP1:90,2] + 31.706;
   1:L PR[91] 10mm/sec CNT100;
   1:  PR[GP1:91,1] = PR[GP1:90,1] + 14.143;
   1:  PR[GP1:91,2] = PR[GP1:90,2] + 29.335;
   1:L PR[91] 10mm/sec CNT100;
   1:  PR[GP1:91,1] = PR[GP1:90,1] + 10.984;
   1:  PR[GP1:91,2] = PR[GP1:90,2] + 26.957;
   1:L PR[91] 10mm/sec CNT100;
   1:  PR[GP1:91,1] = PR[GP1:90,1] + 6.622;
   1:  PR[GP1:91,2] = PR[GP1:90,2] + 23.027;
   1:L PR[91] 10mm/sec CNT100;
   1:  PR[GP1:91,1] = PR[GP1:90,1] + 5.922;
   1:  PR[GP1:91,2] = PR[GP1:90,2] + 21.911;
   1:L PR[91] 10mm/sec CNT100;
   1:  PR[GP1:91,1] = PR[GP1:90,1] + 1.718;
   1:  PR[GP1:91,2] = PR[GP1:90,2] + 16.040;
   1:L PR[91] 10mm/sec CNT100;
   1:  PR[GP1:91,1] = PR[GP1:90,1] + -2.242;
   1:L PR[91] 10mm/sec CNT100;
   1:  PR[GP1:91,1] = PR[GP1:90,1] + -3.450;
   1:  PR[GP1:91,2] = PR[GP1:90,2] + 17.743;
   1:L PR[91] 10mm/sec CNT100;
   1:  PR[GP1:91,1] = PR[GP1:90,1] + -7.096;
   1:  PR[GP1:91,2] = PR[GP1:90,2] + 22.982;
   1:L PR[91] 10mm/sec CNT100;
   1:  PR[GP1:91,1] = PR[GP1:90,1] + -11.491;
   1:  PR[GP1:91,2] = PR[GP1:90,2] + 26.942;
   1:L PR[91] 10mm/sec CNT100;
   1:  PR[GP1:91,1] = PR[GP1:90,1] + -14.646;
   1:  PR[GP1:91,2] = PR[GP1:90,2] + 29.313;
   1:L PR[91] 10mm/sec CNT100;
   1:  PR[GP1:91,1] = PR[GP1:90,1] + -18.867;
   1:  PR[GP1:91,2] = PR[GP1:90,2] + 31.711;
   1:L PR[91] 10mm/sec CNT100;
   1:  PR[GP1:91,1] = PR[GP1:90,1] + -26.788;
   1:  PR[GP1:91,2] = PR[GP1:90,2] + 34.212;
   1:L PR[91] 10mm/sec CNT100;
   1:  PR[GP1:91,1] = PR[GP1:90,1] + -29.362;
   1:  PR[GP1:91,2] = PR[GP1:90,2] + 34.978;
   1:L PR[91] 10mm/sec CNT100;
   1:  PR[GP1:91,1] = PR[GP1:90,1] + -30.920;
   1:  PR[GP1:91,2] = PR[GP1:90,2] + 35.112;
   1:L PR[91] 10mm/sec CNT100;
   1:  PR[GP1:91,1] = PR[GP1:90,1] + -39.638;
   1:  PR[GP1:91,2] = PR[GP1:90,2] + 34.856;
   1:L PR[91] 10mm/sec CNT100;
   1:  PR[GP1:91,1] = PR[GP1:90,1] + -42.417;
   1:  PR[GP1:91,2] = PR[GP1:90,2] + 34.834;
   1:L PR[91] 10mm/sec CNT100;
   1:  PR[GP1:91,1] = PR[GP1:90,1] + -43.175;
   1:  PR[GP1:91,2] = PR[GP1:90,2] + 34.593;
   1:L PR[91] 10mm/sec CNT100;
   1:  PR[GP1:91,1] = PR[GP1:90,1] + -53.891;
   1:  PR[GP1:91,2] = PR[GP1:90,2] + 30.712;
   1:L PR[91] 10mm/sec CNT100;
   1:  PR[GP1:91,1] = PR[GP1:90,1] + -56.995;
   1:  PR[GP1:91,2] = PR[GP1:90,2] + 28.302;
   1:L PR[91] 10mm/sec CNT100;
   1:  PR[GP1:91,1] = PR[GP1:90,1] + -63.450;
   1:  PR[GP1:91,2] = PR[GP1:90,2] + 22.979;
   1:L PR[91] 10mm/sec CNT100;
   1:  PR[GP1:91,1] = PR[GP1:90,1] + -66.528;
   1:  PR[GP1:91,2] = PR[GP1:90,2] + 17.953;
   1:L PR[91] 10mm/sec CNT100;
   1:  PR[GP1:91,1] = PR[GP1:90,1] + -69.795;
   1:  PR[GP1:91,2] = PR[GP1:90,2] + 12.385;
   1:L PR[91] 10mm/sec CNT100;
   1:  PR[GP1:91,1] = PR[GP1:90,1] + -71.047;
   1:  PR[GP1:91,2] = PR[GP1:90,2] + 5.684;
   1:L PR[91] 10mm/sec CNT100;
   1:  PR[GP1:91,1] = PR[GP1:90,1] + -71.193;
   1:  PR[GP1:91,2] = PR[GP1:90,2] + 5.006;
   1:L PR[91] 10mm/sec CNT100;
   1:  PR[GP1:91,1] = PR[GP1:90,1] + -72.040;
   1:  PR[GP1:91,2] = PR[GP1:90,2] + 0.282;
   1:L PR[91] 10mm/sec CNT100;
   1:  PR[GP1:91,1] = PR[GP1:90,1] + -70.742;
   1:  PR[GP1:91,2] = PR[GP1:90,2] + -6.519;
   1:L PR[91] 10mm/sec CNT100;
   1:  PR[GP1:91,1] = PR[GP1:90,1] + -69.793;
   1:  PR[GP1:91,2] = PR[GP1:90,2] + -11.829;
   1:L PR[91] 10mm/sec CNT100;
   1:  PR[GP1:91,1] = PR[GP1:90,1] + -66.528;
   1:  PR[GP1:91,2] = PR[GP1:90,2] + -17.395;
   1:L PR[91] 10mm/sec CNT100;
   1:  PR[GP1:91,1] = PR[GP1:90,1] + -63.450;
   1:  PR[GP1:91,2] = PR[GP1:90,2] + -22.421;
   1:L PR[91] 10mm/sec CNT100;
   1:  PR[GP1:91,1] = PR[GP1:90,1] + -56.995;
   1:  PR[GP1:91,2] = PR[GP1:90,2] + -27.743;
   1:L PR[91] 10mm/sec CNT100;
   1:  PR[GP1:91,1] = PR[GP1:90,1] + -53.891;
   1:  PR[GP1:91,2] = PR[GP1:90,2] + -30.154;
   1:L PR[91] 10mm/sec CNT100;
   1:  PR[GP1:91,1] = PR[GP1:90,1] + -43.175;
   1:  PR[GP1:91,2] = PR[GP1:90,2] + -34.035;
   1:L PR[91] 10mm/sec CNT100;
   1:  PR[GP1:91,1] = PR[GP1:90,1] + -42.417;
   1:  PR[GP1:91,2] = PR[GP1:90,2] + -34.275;
   1:L PR[91] 10mm/sec CNT100;
   1:  PR[GP1:91,1] = PR[GP1:90,1] + -39.638;
   1:  PR[GP1:91,2] = PR[GP1:90,2] + -34.298;
   1:L PR[91] 10mm/sec CNT100;
   1:  PR[GP1:91,1] = PR[GP1:90,1] + -30.920;
   1:  PR[GP1:91,2] = PR[GP1:90,2] + -34.553;
   1:L PR[91] 10mm/sec CNT100;
   1:  PR[GP1:91,1] = PR[GP1:90,1] + -29.368;
   1:  PR[GP1:91,2] = PR[GP1:90,2] + -34.421;
   1:L PR[91] 10mm/sec CNT100;
   1:  PR[GP1:91,1] = PR[GP1:90,1] + -21.823;
   1:  PR[GP1:91,2] = PR[GP1:90,2] + -32.003;
   1:L PR[91] 10mm/sec CNT100;
   1:  PR[GP1:91,1] = PR[GP1:90,1] + -18.860;
   1:  PR[GP1:91,2] = PR[GP1:90,2] + -31.150;
   1:L PR[91] 10mm/sec CNT100;
   1:  PR[GP1:91,1] = PR[GP1:90,1] + -14.646;
   1:  PR[GP1:91,2] = PR[GP1:90,2] + -28.755;
   1:L PR[91] 10mm/sec CNT100;
   1:  PR[GP1:91,1] = PR[GP1:90,1] + -11.491;
   1:  PR[GP1:91,2] = PR[GP1:90,2] + -26.384;
   1:L PR[91] 10mm/sec CNT100;
   1:  PR[GP1:91,1] = PR[GP1:90,1] + -7.107;
   1:  PR[GP1:91,2] = PR[GP1:90,2] + -22.434;
   1:L PR[91] 10mm/sec CNT100;
   1:  PR[GP1:91,1] = PR[GP1:90,1] + -6.414;
   1:  PR[GP1:91,2] = PR[GP1:90,2] + -21.328;
   1:L PR[91] 10mm/sec CNT100;
   1:  PR[GP1:91,1] = PR[GP1:90,1] + -2.241;
   1:  PR[GP1:91,2] = PR[GP1:90,2] + -15.482;
   1:L PR[91] 10mm/sec CNT100;
   1:  PR[GP1:91,1] = PR[GP1:90,1] + 1.719;
   1:L PR[91] 10mm/sec CNT100;
   1:  PR[GP1:91,1] = PR[GP1:90,1] + 5.160;
   1:  PR[GP1:91,2] = PR[GP1:90,2] + -20.765;
   1:  PR[GP1:91,3] = PR[GP1:90,3] + 37.515;
   1:L PR[91] 10mm/sec CNT100;
   1:  PR[GP1:91,1] = PR[GP1:90,1] + 6.341;
   1:  PR[GP1:91,2] = PR[GP1:90,2] + -22.458;
   1:L PR[91] 10mm/sec CNT100;
   1:  PR[GP1:91,1] = PR[GP1:90,1] + 11.154;
   1:  PR[GP1:91,2] = PR[GP1:90,2] + -26.794;
   1:L PR[91] 10mm/sec CNT100;
   1:  PR[GP1:91,1] = PR[GP1:90,1] + 13.501;
   1:  PR[GP1:91,2] = PR[GP1:90,2] + -28.561;
   1:L PR[91] 10mm/sec CNT100;
   1:  PR[GP1:91,1] = PR[GP1:90,1] + 18.306;
   1:  PR[GP1:91,2] = PR[GP1:90,2] + -31.284;
   1:L PR[91] 10mm/sec CNT100;
   1:  PR[GP1:91,1] = PR[GP1:90,1] + 25.071;
   1:  PR[GP1:91,2] = PR[GP1:90,2] + -33.420;
   1:L PR[91] 10mm/sec CNT100;
   1:  PR[GP1:91,1] = PR[GP1:90,1] + 28.495;
   1:  PR[GP1:91,2] = PR[GP1:90,2] + -34.438;
   1:L PR[91] 10mm/sec CNT100;
   1:  PR[GP1:91,1] = PR[GP1:90,1] + 30.577;
   1:  PR[GP1:91,2] = PR[GP1:90,2] + -34.618;
   1:L PR[91] 10mm/sec CNT100;
   1:  PR[GP1:91,1] = PR[GP1:90,1] + 41.814;
   1:  PR[GP1:91,2] = PR[GP1:90,2] + -34.290;
   1:L PR[91] 10mm/sec CNT100;
   1:  PR[GP1:91,1] = PR[GP1:90,1] + 53.307;
   1:  PR[GP1:91,2] = PR[GP1:90,2] + -30.138;
   1:L PR[91] 10mm/sec CNT100;
   1:  PR[GP1:91,1] = PR[GP1:90,1] + 55.743;
   1:  PR[GP1:91,2] = PR[GP1:90,2] + -28.246;
   1:L PR[91] 10mm/sec CNT100;
   1:  PR[GP1:91,1] = PR[GP1:90,1] + 62.835;
   1:  PR[GP1:91,2] = PR[GP1:90,2] + -22.390;
   1:L PR[91] 10mm/sec CNT100;
   1:  PR[GP1:91,1] = PR[GP1:90,1] + 65.516;
   1:  PR[GP1:91,2] = PR[GP1:90,2] + -18.019;
   1:L PR[91] 10mm/sec CNT100;
   1:  PR[GP1:91,1] = PR[GP1:90,1] + 69.159;
   1:  PR[GP1:91,2] = PR[GP1:90,2] + -11.827;
   1:L PR[91] 10mm/sec CNT100;
   1:  PR[GP1:91,1] = PR[GP1:90,1] + 70.283;
   1:  PR[GP1:91,2] = PR[GP1:90,2] + -5.806;
   1:L PR[91] 10mm/sec CNT100;
   1:  PR[GP1:91,1] = PR[GP1:90,1] + 70.415;
   1:  PR[GP1:91,2] = PR[GP1:90,2] + -5.196;
   1:L PR[91] 10mm/sec CNT100;
   1:  PR[GP1:91,1] = PR[GP1:90,1] + 71.394;
   1:  PR[GP1:91,2] = PR[GP1:90,2] + 0.276;
   1:L PR[91] 10mm/sec CNT100;
   1:  PR[GP1:91,1] = PR[GP1:90,1] + 70.216;
   1:  PR[GP1:91,2] = PR[GP1:90,2] + 6.455;
   1:L PR[91] 10mm/sec CNT100;
   1:  PR[GP1:91,1] = PR[GP1:90,1] + 69.158;
   1:  PR[GP1:91,2] = PR[GP1:90,2] + 12.387;
   1:L PR[91] 10mm/sec CNT100;
   1:  PR[GP1:91,1] = PR[GP1:90,1] + 65.516;
   1:  PR[GP1:91,2] = PR[GP1:90,2] + 18.577;
   1:L PR[91] 10mm/sec CNT100;
   1:  PR[GP1:91,1] = PR[GP1:90,1] + 62.835;
   1:  PR[GP1:91,2] = PR[GP1:90,2] + 22.948;
   1:L PR[91] 10mm/sec CNT100;
   1:  PR[GP1:91,1] = PR[GP1:90,1] + 55.743;
   1:  PR[GP1:91,2] = PR[GP1:90,2] + 28.804;
   1:L PR[91] 10mm/sec CNT100;
   1:  PR[GP1:91,1] = PR[GP1:90,1] + 53.307;
   1:  PR[GP1:91,2] = PR[GP1:90,2] + 30.697;
   1:L PR[91] 10mm/sec CNT100;
   1:  PR[GP1:91,1] = PR[GP1:90,1] + 41.846;
   1:  PR[GP1:91,2] = PR[GP1:90,2] + 34.844;
   1:L PR[91] 10mm/sec CNT100;
   1:  PR[GP1:91,1] = PR[GP1:90,1] + 30.577;
   1:  PR[GP1:91,2] = PR[GP1:90,2] + 35.176;
   1:L PR[91] 10mm/sec CNT100;
   1:  PR[GP1:91,1] = PR[GP1:90,1] + 28.501;
   1:  PR[GP1:91,2] = PR[GP1:90,2] + 34.997;
   1:L PR[91] 10mm/sec CNT100;
   1:  PR[GP1:91,1] = PR[GP1:90,1] + 21.702;
   1:  PR[GP1:91,2] = PR[GP1:90,2] + 32.819;
   1:L PR[91] 10mm/sec CNT100;
   1:  PR[GP1:91,1] = PR[GP1:90,1] + 18.300;
   1:  PR[GP1:91,2] = PR[GP1:90,2] + 31.838;
   1:L PR[91] 10mm/sec CNT100;
   1:  PR[GP1:91,1] = PR[GP1:90,1] + 13.501;
   1:  PR[GP1:91,2] = PR[GP1:90,2] + 29.119;
   1:L PR[91] 10mm/sec CNT100;
   1:  PR[GP1:91,1] = PR[GP1:90,1] + 11.154;
   1:  PR[GP1:91,2] = PR[GP1:90,2] + 27.353;
   1:L PR[91] 10mm/sec CNT100;
   1:  PR[GP1:91,1] = PR[GP1:90,1] + 6.352;
   1:  PR[GP1:91,2] = PR[GP1:90,2] + 23.026;
   1:L PR[91] 10mm/sec CNT100;
   1:  PR[GP1:91,1] = PR[GP1:90,1] + 6.147;
   1:  PR[GP1:91,2] = PR[GP1:90,2] + 22.698;
   1:L PR[91] 10mm/sec CNT100;
   1:  PR[GP1:91,1] = PR[GP1:90,1] + 1.633;
   1:  PR[GP1:91,2] = PR[GP1:90,2] + 16.365;
   1:L PR[91] 10mm/sec CNT100;
   1:  PR[GP1:91,1] = PR[GP1:90,1] + -2.155;
   1:L PR[91] 10mm/sec CNT100;
   1:  PR[GP1:91,1] = PR[GP1:90,1] + -5.687;
   1:  PR[GP1:91,2] = PR[GP1:90,2] + 21.345;
   1:L PR[91] 10mm/sec CNT100;
   1:  PR[GP1:91,1] = PR[GP1:90,1] + -6.822;
   1:  PR[GP1:91,2] = PR[GP1:90,2] + 22.976;
   1:L PR[91] 10mm/sec CNT100;
   1:  PR[GP1:91,1] = PR[GP1:90,1] + -11.659;
   1:  PR[GP1:91,2] = PR[GP1:90,2] + 27.335;
   1:L PR[91] 10mm/sec CNT100;
   1:  PR[GP1:91,1] = PR[GP1:90,1] + -14.000;
   1:  PR[GP1:91,2] = PR[GP1:90,2] + 29.094;
   1:L PR[91] 10mm/sec CNT100;
   1:  PR[GP1:91,1] = PR[GP1:90,1] + -18.840;
   1:  PR[GP1:91,2] = PR[GP1:90,2] + 31.844;
   1:L PR[91] 10mm/sec CNT100;
   1:  PR[GP1:91,1] = PR[GP1:90,1] + -25.606;
   1:  PR[GP1:91,2] = PR[GP1:90,2] + 33.980;
   1:L PR[91] 10mm/sec CNT100;
   1:  PR[GP1:91,1] = PR[GP1:90,1] + -29.024;
   1:  PR[GP1:91,2] = PR[GP1:90,2] + 34.997;
   1:L PR[91] 10mm/sec CNT100;
   1:  PR[GP1:91,1] = PR[GP1:90,1] + -31.111;
   1:  PR[GP1:91,2] = PR[GP1:90,2] + 35.176;
   1:L PR[91] 10mm/sec CNT100;
   1:  PR[GP1:91,1] = PR[GP1:90,1] + -42.346;
   1:  PR[GP1:91,2] = PR[GP1:90,2] + 34.847;
   1:L PR[91] 10mm/sec CNT100;
   1:  PR[GP1:91,1] = PR[GP1:90,1] + -53.837;
   1:  PR[GP1:91,2] = PR[GP1:90,2] + 30.692;
   1:L PR[91] 10mm/sec CNT100;
   1:  PR[GP1:91,1] = PR[GP1:90,1] + -56.273;
   1:  PR[GP1:91,2] = PR[GP1:90,2] + 28.799;
   1:L PR[91] 10mm/sec CNT100;
   1:  PR[GP1:91,1] = PR[GP1:90,1] + -63.363;
   1:  PR[GP1:91,2] = PR[GP1:90,2] + 22.953;
   1:L PR[91] 10mm/sec CNT100;
   1:  PR[GP1:91,1] = PR[GP1:90,1] + -66.043;
   1:  PR[GP1:91,2] = PR[GP1:90,2] + 18.576;
   1:L PR[91] 10mm/sec CNT100;
   1:  PR[GP1:91,1] = PR[GP1:90,1] + -69.686;
   1:  PR[GP1:91,2] = PR[GP1:90,2] + 12.368;
   1:L PR[91] 10mm/sec CNT100;
   1:  PR[GP1:91,1] = PR[GP1:90,1] + -70.810;
   1:  PR[GP1:91,2] = PR[GP1:90,2] + 6.353;
   1:L PR[91] 10mm/sec CNT100;
   1:  PR[GP1:91,1] = PR[GP1:90,1] + -70.941;
   1:  PR[GP1:91,2] = PR[GP1:90,2] + 5.744;
   1:L PR[91] 10mm/sec CNT100;
   1:  PR[GP1:91,1] = PR[GP1:90,1] + -71.921;
   1:  PR[GP1:91,2] = PR[GP1:90,2] + 0.282;
   1:L PR[91] 10mm/sec CNT100;
   1:  PR[GP1:91,1] = PR[GP1:90,1] + -70.743;
   1:  PR[GP1:91,2] = PR[GP1:90,2] + -5.891;
   1:L PR[91] 10mm/sec CNT100;
   1:  PR[GP1:91,1] = PR[GP1:90,1] + -69.685;
   1:  PR[GP1:91,2] = PR[GP1:90,2] + -11.812;
   1:L PR[91] 10mm/sec CNT100;
   1:  PR[GP1:91,1] = PR[GP1:90,1] + -66.043;
   1:  PR[GP1:91,2] = PR[GP1:90,2] + -18.018;
   1:L PR[91] 10mm/sec CNT100;
   1:  PR[GP1:91,1] = PR[GP1:90,1] + -63.363;
   1:  PR[GP1:91,2] = PR[GP1:90,2] + -22.395;
   1:L PR[91] 10mm/sec CNT100;
   1:  PR[GP1:91,1] = PR[GP1:90,1] + -56.273;
   1:  PR[GP1:91,2] = PR[GP1:90,2] + -28.241;
   1:L PR[91] 10mm/sec CNT100;
   1:  PR[GP1:91,1] = PR[GP1:90,1] + -53.837;
   1:  PR[GP1:91,2] = PR[GP1:90,2] + -30.134;
   1:L PR[91] 10mm/sec CNT100;
   1:  PR[GP1:91,1] = PR[GP1:90,1] + -42.377;
   1:  PR[GP1:91,2] = PR[GP1:90,2] + -34.285;
   1:L PR[91] 10mm/sec CNT100;
   1:  PR[GP1:91,1] = PR[GP1:90,1] + -31.111;
   1:  PR[GP1:91,2] = PR[GP1:90,2] + -34.618;
   1:L PR[91] 10mm/sec CNT100;
   1:  PR[GP1:91,1] = PR[GP1:90,1] + -29.031;
   1:  PR[GP1:91,2] = PR[GP1:90,2] + -34.440;
   1:L PR[91] 10mm/sec CNT100;
   1:  PR[GP1:91,1] = PR[GP1:90,1] + -22.230;
   1:  PR[GP1:91,2] = PR[GP1:90,2] + -32.261;
   1:L PR[91] 10mm/sec CNT100;
   1:  PR[GP1:91,1] = PR[GP1:90,1] + -18.833;
   1:  PR[GP1:91,2] = PR[GP1:90,2] + -31.282;
   1:L PR[91] 10mm/sec CNT100;
   1:  PR[GP1:91,1] = PR[GP1:90,1] + -14.000;
   1:  PR[GP1:91,2] = PR[GP1:90,2] + -28.536;
   1:L PR[91] 10mm/sec CNT100;
   1:  PR[GP1:91,1] = PR[GP1:90,1] + -11.659;
   1:  PR[GP1:91,2] = PR[GP1:90,2] + -26.777;
   1:L PR[91] 10mm/sec CNT100;
   1:  PR[GP1:91,1] = PR[GP1:90,1] + -6.832;
   1:  PR[GP1:91,2] = PR[GP1:90,2] + -22.427;
   1:L PR[91] 10mm/sec CNT100;
   1:  PR[GP1:91,1] = PR[GP1:90,1] + -6.636;
   1:  PR[GP1:91,2] = PR[GP1:90,2] + -22.114;
   1:L PR[91] 10mm/sec CNT100;
   1:  PR[GP1:91,1] = PR[GP1:90,1] + -2.155;
   1:  PR[GP1:91,2] = PR[GP1:90,2] + -15.807;
   1:L PR[91] 10mm/sec CNT100;
   1:  PR[GP1:91,1] = PR[GP1:90,1] + 1.633;
   1:L PR[91] 10mm/sec CNT100;
   1:  PR[GP1:91,1] = PR[GP1:90,1] + 6.012;
   1:  PR[GP1:91,2] = PR[GP1:90,2] + -22.409;
   1:  PR[GP1:91,3] = PR[GP1:90,3] + 38.125;
   1:L PR[91] 10mm/sec CNT100;
   1:  PR[GP1:91,1] = PR[GP1:90,1] + 6.073;
   1:  PR[GP1:91,2] = PR[GP1:90,2] + -22.483;
   1:L PR[91] 10mm/sec CNT100;
   1:  PR[GP1:91,1] = PR[GP1:90,1] + 7.306;
   1:  PR[GP1:91,2] = PR[GP1:90,2] + -23.569;
   1:L PR[91] 10mm/sec CNT100;
   1:  PR[GP1:91,1] = PR[GP1:90,1] + 11.325;
   1:  PR[GP1:91,2] = PR[GP1:90,2] + -27.190;
   1:L PR[91] 10mm/sec CNT100;
   1:  PR[GP1:91,1] = PR[GP1:90,1] + 12.859;
   1:  PR[GP1:91,2] = PR[GP1:90,2] + -28.344;
   1:L PR[91] 10mm/sec CNT100;
   1:  PR[GP1:91,1] = PR[GP1:90,1] + 18.279;
   1:  PR[GP1:91,2] = PR[GP1:90,2] + -31.416;
   1:L PR[91] 10mm/sec CNT100;
   1:  PR[GP1:91,1] = PR[GP1:90,1] + 23.889;
   1:  PR[GP1:91,2] = PR[GP1:90,2] + -33.187;
   1:L PR[91] 10mm/sec CNT100;
   1:  PR[GP1:91,1] = PR[GP1:90,1] + 28.158;
   1:  PR[GP1:91,2] = PR[GP1:90,2] + -34.458;
   1:L PR[91] 10mm/sec CNT100;
   1:  PR[GP1:91,1] = PR[GP1:90,1] + 30.768;
   1:  PR[GP1:91,2] = PR[GP1:90,2] + -34.682;
   1:L PR[91] 10mm/sec CNT100;
   1:  PR[GP1:91,1] = PR[GP1:90,1] + 41.174;
   1:  PR[GP1:91,2] = PR[GP1:90,2] + -34.378;
   1:L PR[91] 10mm/sec CNT100;
   1:  PR[GP1:91,1] = PR[GP1:90,1] + 41.736;
   1:  PR[GP1:91,2] = PR[GP1:90,2] + -34.308;
   1:L PR[91] 10mm/sec CNT100;
   1:  PR[GP1:91,1] = PR[GP1:90,1] + 44.898;
   1:  PR[GP1:91,2] = PR[GP1:90,2] + -33.140;
   1:L PR[91] 10mm/sec CNT100;
   1:  PR[GP1:91,1] = PR[GP1:90,1] + 53.252;
   1:  PR[GP1:91,2] = PR[GP1:90,2] + -30.118;
   1:L PR[91] 10mm/sec CNT100;
   1:  PR[GP1:91,1] = PR[GP1:90,1] + 55.021;
   1:  PR[GP1:91,2] = PR[GP1:90,2] + -28.744;
   1:L PR[91] 10mm/sec CNT100;
   1:  PR[GP1:91,1] = PR[GP1:90,1] + 62.748;
   1:  PR[GP1:91,2] = PR[GP1:90,2] + -22.364;
   1:L PR[91] 10mm/sec CNT100;
   1:  PR[GP1:91,1] = PR[GP1:90,1] + 65.032;
   1:  PR[GP1:91,2] = PR[GP1:90,2] + -18.640;
   1:L PR[91] 10mm/sec CNT100;
   1:  PR[GP1:91,1] = PR[GP1:90,1] + 69.051;
   1:  PR[GP1:91,2] = PR[GP1:90,2] + -11.811;
   1:L PR[91] 10mm/sec CNT100;
   1:  PR[GP1:91,1] = PR[GP1:90,1] + 70.047;
   1:  PR[GP1:91,2] = PR[GP1:90,2] + -6.476;
   1:L PR[91] 10mm/sec CNT100;
   1:  PR[GP1:91,1] = PR[GP1:90,1] + 70.163;
   1:  PR[GP1:91,2] = PR[GP1:90,2] + -5.935;
   1:L PR[91] 10mm/sec CNT100;
   1:  PR[GP1:91,1] = PR[GP1:90,1] + 71.275;
   1:  PR[GP1:91,2] = PR[GP1:90,2] + 0.276;
   1:L PR[91] 10mm/sec CNT100;
   1:  PR[GP1:91,1] = PR[GP1:90,1] + 70.217;
   1:  PR[GP1:91,2] = PR[GP1:90,2] + 5.826;
   1:L PR[91] 10mm/sec CNT100;
   1:  PR[GP1:91,1] = PR[GP1:90,1] + 69.049;
   1:  PR[GP1:91,2] = PR[GP1:90,2] + 12.371;
   1:L PR[91] 10mm/sec CNT100;
   1:  PR[GP1:91,1] = PR[GP1:90,1] + 65.032;
   1:  PR[GP1:91,2] = PR[GP1:90,2] + 19.198;
   1:L PR[91] 10mm/sec CNT100;
   1:  PR[GP1:91,1] = PR[GP1:90,1] + 62.748;
   1:  PR[GP1:91,2] = PR[GP1:90,2] + 22.922;
   1:L PR[91] 10mm/sec CNT100;
   1:  PR[GP1:91,1] = PR[GP1:90,1] + 55.021;
   1:  PR[GP1:91,2] = PR[GP1:90,2] + 29.302;
   1:L PR[91] 10mm/sec CNT100;
   1:  PR[GP1:91,1] = PR[GP1:90,1] + 53.252;
   1:  PR[GP1:91,2] = PR[GP1:90,2] + 30.676;
   1:L PR[91] 10mm/sec CNT100;
   1:  PR[GP1:91,1] = PR[GP1:90,1] + 44.898;
   1:  PR[GP1:91,2] = PR[GP1:90,2] + 33.698;
   1:L PR[91] 10mm/sec CNT100;
   1:  PR[GP1:91,1] = PR[GP1:90,1] + 41.736;
   1:  PR[GP1:91,2] = PR[GP1:90,2] + 34.866;
   1:L PR[91] 10mm/sec CNT100;
   1:  PR[GP1:91,1] = PR[GP1:90,1] + 41.174;
   1:  PR[GP1:91,2] = PR[GP1:90,2] + 34.936;
   1:L PR[91] 10mm/sec CNT100;
   1:  PR[GP1:91,1] = PR[GP1:90,1] + 30.768;
   1:  PR[GP1:91,2] = PR[GP1:90,2] + 35.240;
   1:L PR[91] 10mm/sec CNT100;
   1:  PR[GP1:91,1] = PR[GP1:90,1] + 28.165;
   1:  PR[GP1:91,2] = PR[GP1:90,2] + 35.016;
   1:L PR[91] 10mm/sec CNT100;
   1:  PR[GP1:91,1] = PR[GP1:90,1] + 22.109;
   1:  PR[GP1:91,2] = PR[GP1:90,2] + 33.076;
   1:L PR[91] 10mm/sec CNT100;
   1:  PR[GP1:91,1] = PR[GP1:90,1] + 18.272;
   1:  PR[GP1:91,2] = PR[GP1:90,2] + 31.970;
   1:L PR[91] 10mm/sec CNT100;
   1:  PR[GP1:91,1] = PR[GP1:90,1] + 12.859;
   1:  PR[GP1:91,2] = PR[GP1:90,2] + 28.902;
   1:L PR[91] 10mm/sec CNT100;
   1:  PR[GP1:91,1] = PR[GP1:90,1] + 11.325;
   1:  PR[GP1:91,2] = PR[GP1:90,2] + 27.748;
   1:L PR[91] 10mm/sec CNT100;
   1:  PR[GP1:91,1] = PR[GP1:90,1] + 7.306;
   1:  PR[GP1:91,2] = PR[GP1:90,2] + 24.127;
   1:L PR[91] 10mm/sec CNT100;
   1:  PR[GP1:91,1] = PR[GP1:90,1] + 6.073;
   1:  PR[GP1:91,2] = PR[GP1:90,2] + 23.041;
   1:L PR[91] 10mm/sec CNT100;
   1:  PR[GP1:91,1] = PR[GP1:90,1] + 6.010;
   1:  PR[GP1:91,2] = PR[GP1:90,2] + 22.964;
   1:L PR[91] 10mm/sec CNT100;
   1:  PR[GP1:91,1] = PR[GP1:90,1] + 1.547;
   1:  PR[GP1:91,2] = PR[GP1:90,2] + 16.690;
   1:L PR[91] 10mm/sec CNT100;
   1:  PR[GP1:91,1] = PR[GP1:90,1] + -2.068;
   1:L PR[91] 10mm/sec CNT100;
   1:  PR[GP1:91,1] = PR[GP1:90,1] + -6.487;
   1:  PR[GP1:91,2] = PR[GP1:90,2] + 22.922;
   1:L PR[91] 10mm/sec CNT100;
   1:  PR[GP1:91,1] = PR[GP1:90,1] + -6.552;
   1:  PR[GP1:91,2] = PR[GP1:90,2] + 23.000;
   1:L PR[91] 10mm/sec CNT100;
   1:  PR[GP1:91,1] = PR[GP1:90,1] + -7.832;
   1:  PR[GP1:91,2] = PR[GP1:90,2] + 24.127;
   1:L PR[91] 10mm/sec CNT100;
   1:  PR[GP1:91,1] = PR[GP1:90,1] + -11.827;
   1:  PR[GP1:91,2] = PR[GP1:90,2] + 27.727;
   1:L PR[91] 10mm/sec CNT100;
   1:  PR[GP1:91,1] = PR[GP1:90,1] + -13.354;
   1:  PR[GP1:91,2] = PR[GP1:90,2] + 28.874;
   1:L PR[91] 10mm/sec CNT100;
   1:  PR[GP1:91,1] = PR[GP1:90,1] + -18.812;
   1:  PR[GP1:91,2] = PR[GP1:90,2] + 31.976;
   1:L PR[91] 10mm/sec CNT100;
   1:  PR[GP1:91,1] = PR[GP1:90,1] + -24.425;
   1:  PR[GP1:91,2] = PR[GP1:90,2] + 33.748;
   1:L PR[91] 10mm/sec CNT100;
   1:  PR[GP1:91,1] = PR[GP1:90,1] + -28.687;
   1:  PR[GP1:91,2] = PR[GP1:90,2] + 35.016;
   1:L PR[91] 10mm/sec CNT100;
   1:  PR[GP1:91,1] = PR[GP1:90,1] + -31.303;
   1:  PR[GP1:91,2] = PR[GP1:90,2] + 35.240;
   1:L PR[91] 10mm/sec CNT100;
   1:  PR[GP1:91,1] = PR[GP1:90,1] + -41.707;
   1:  PR[GP1:91,2] = PR[GP1:90,2] + 34.936;
   1:L PR[91] 10mm/sec CNT100;
   1:  PR[GP1:91,1] = PR[GP1:90,1] + -42.269;
   1:  PR[GP1:91,2] = PR[GP1:90,2] + 34.865;
   1:L PR[91] 10mm/sec CNT100;
   1:  PR[GP1:91,1] = PR[GP1:90,1] + -45.424;
   1:  PR[GP1:91,2] = PR[GP1:90,2] + 33.698;
   1:L PR[91] 10mm/sec CNT100;
   1:  PR[GP1:91,1] = PR[GP1:90,1] + -53.782;
   1:  PR[GP1:91,2] = PR[GP1:90,2] + 30.671;
   1:L PR[91] 10mm/sec CNT100;
   1:  PR[GP1:91,1] = PR[GP1:90,1] + -55.551;
   1:  PR[GP1:91,2] = PR[GP1:90,2] + 29.297;
   1:L PR[91] 10mm/sec CNT100;
   1:  PR[GP1:91,1] = PR[GP1:90,1] + -63.277;
   1:  PR[GP1:91,2] = PR[GP1:90,2] + 22.927;
   1:L PR[91] 10mm/sec CNT100;
   1:  PR[GP1:91,1] = PR[GP1:90,1] + -65.559;
   1:  PR[GP1:91,2] = PR[GP1:90,2] + 19.199;
   1:L PR[91] 10mm/sec CNT100;
   1:  PR[GP1:91,1] = PR[GP1:90,1] + -69.578;
   1:  PR[GP1:91,2] = PR[GP1:90,2] + 12.351;
   1:L PR[91] 10mm/sec CNT100;
   1:  PR[GP1:91,1] = PR[GP1:90,1] + -70.573;
   1:  PR[GP1:91,2] = PR[GP1:90,2] + 7.022;
   1:L PR[91] 10mm/sec CNT100;
   1:  PR[GP1:91,1] = PR[GP1:90,1] + -70.690;
   1:  PR[GP1:91,2] = PR[GP1:90,2] + 6.481;
   1:L PR[91] 10mm/sec CNT100;
   1:  PR[GP1:91,1] = PR[GP1:90,1] + -71.802;
   1:  PR[GP1:91,2] = PR[GP1:90,2] + 0.282;
   1:L PR[91] 10mm/sec CNT100;
   1:  PR[GP1:91,1] = PR[GP1:90,1] + -70.743;
   1:  PR[GP1:91,2] = PR[GP1:90,2] + -5.262;
   1:L PR[91] 10mm/sec CNT100;
   1:  PR[GP1:91,1] = PR[GP1:90,1] + -69.576;
   1:  PR[GP1:91,2] = PR[GP1:90,2] + -11.795;
   1:L PR[91] 10mm/sec CNT100;
   1:  PR[GP1:91,1] = PR[GP1:90,1] + -65.559;
   1:  PR[GP1:91,2] = PR[GP1:90,2] + -18.641;
   1:L PR[91] 10mm/sec CNT100;
   1:  PR[GP1:91,1] = PR[GP1:90,1] + -63.277;
   1:  PR[GP1:91,2] = PR[GP1:90,2] + -22.369;
   1:L PR[91] 10mm/sec CNT100;
   1:  PR[GP1:91,1] = PR[GP1:90,1] + -55.551;
   1:  PR[GP1:91,2] = PR[GP1:90,2] + -28.739;
   1:L PR[91] 10mm/sec CNT100;
   1:  PR[GP1:91,1] = PR[GP1:90,1] + -53.782;
   1:  PR[GP1:91,2] = PR[GP1:90,2] + -30.113;
   1:L PR[91] 10mm/sec CNT100;
   1:  PR[GP1:91,1] = PR[GP1:90,1] + -45.424;
   1:  PR[GP1:91,2] = PR[GP1:90,2] + -33.140;
   1:L PR[91] 10mm/sec CNT100;
   1:  PR[GP1:91,1] = PR[GP1:90,1] + -42.269;
   1:  PR[GP1:91,2] = PR[GP1:90,2] + -34.307;
   1:L PR[91] 10mm/sec CNT100;
   1:  PR[GP1:91,1] = PR[GP1:90,1] + -41.707;
   1:  PR[GP1:91,2] = PR[GP1:90,2] + -34.377;
   1:L PR[91] 10mm/sec CNT100;
   1:  PR[GP1:91,1] = PR[GP1:90,1] + -31.303;
   1:  PR[GP1:91,2] = PR[GP1:90,2] + -34.682;
   1:L PR[91] 10mm/sec CNT100;
   1:  PR[GP1:91,1] = PR[GP1:90,1] + -28.693;
   1:  PR[GP1:91,2] = PR[GP1:90,2] + -34.459;
   1:L PR[91] 10mm/sec CNT100;
   1:  PR[GP1:91,1] = PR[GP1:90,1] + -22.637;
   1:  PR[GP1:91,2] = PR[GP1:90,2] + -32.519;
   1:L PR[91] 10mm/sec CNT100;
   1:  PR[GP1:91,1] = PR[GP1:90,1] + -18.806;
   1:  PR[GP1:91,2] = PR[GP1:90,2] + -31.415;
   1:L PR[91] 10mm/sec CNT100;
   1:  PR[GP1:91,1] = PR[GP1:90,1] + -13.354;
   1:  PR[GP1:91,2] = PR[GP1:90,2] + -28.316;
   1:L PR[91] 10mm/sec CNT100;
   1:  PR[GP1:91,1] = PR[GP1:90,1] + -11.827;
   1:  PR[GP1:91,2] = PR[GP1:90,2] + -27.169;
   1:L PR[91] 10mm/sec CNT100;
   1:  PR[GP1:91,1] = PR[GP1:90,1] + -7.832;
   1:  PR[GP1:91,2] = PR[GP1:90,2] + -23.569;
   1:L PR[91] 10mm/sec CNT100;
   1:  PR[GP1:91,1] = PR[GP1:90,1] + -6.552;
   1:  PR[GP1:91,2] = PR[GP1:90,2] + -22.443;
   1:L PR[91] 10mm/sec CNT100;
   1:  PR[GP1:91,1] = PR[GP1:90,1] + -6.488;
   1:  PR[GP1:91,2] = PR[GP1:90,2] + -22.364;
   1:L PR[91] 10mm/sec CNT100;
   1:  PR[GP1:91,1] = PR[GP1:90,1] + -2.068;
   1:  PR[GP1:91,2] = PR[GP1:90,2] + -16.132;
   1:L PR[91] 10mm/sec CNT100;
   1:  PR[GP1:91,1] = PR[GP1:90,1] + 1.547;
   1:L PR[91] 10mm/sec CNT100;
   1:  PR[GP1:91,1] = PR[GP1:90,1] + 5.579;
   1:  PR[GP1:91,2] = PR[GP1:90,2] + -22.246;
   1:  PR[GP1:91,3] = PR[GP1:90,3] + 38.735;
   1:L PR[91] 10mm/sec CNT100;
   1:  PR[GP1:91,1] = PR[GP1:90,1] + 5.846;
   1:  PR[GP1:91,2] = PR[GP1:90,2] + -22.570;
   1:L PR[91] 10mm/sec CNT100;
   1:  PR[GP1:91,1] = PR[GP1:90,1] + 9.543;
   1:  PR[GP1:91,2] = PR[GP1:90,2] + -25.826;
   1:L PR[91] 10mm/sec CNT100;
   1:  PR[GP1:91,1] = PR[GP1:90,1] + 11.495;
   1:  PR[GP1:91,2] = PR[GP1:90,2] + -27.585;
   1:L PR[91] 10mm/sec CNT100;
   1:  PR[GP1:91,1] = PR[GP1:90,1] + 12.217;
   1:  PR[GP1:91,2] = PR[GP1:90,2] + -28.128;
   1:L PR[91] 10mm/sec CNT100;
   1:  PR[GP1:91,1] = PR[GP1:90,1] + 18.252;
   1:  PR[GP1:91,2] = PR[GP1:90,2] + -31.548;
   1:L PR[91] 10mm/sec CNT100;
   1:  PR[GP1:91,1] = PR[GP1:90,1] + 22.707;
   1:  PR[GP1:91,2] = PR[GP1:90,2] + -32.955;
   1:L PR[91] 10mm/sec CNT100;
   1:  PR[GP1:91,1] = PR[GP1:90,1] + 27.822;
   1:  PR[GP1:91,2] = PR[GP1:90,2] + -34.477;
   1:L PR[91] 10mm/sec CNT100;
   1:  PR[GP1:91,1] = PR[GP1:90,1] + 30.959;
   1:  PR[GP1:91,2] = PR[GP1:90,2] + -34.747;
   1:L PR[91] 10mm/sec CNT100;
   1:  PR[GP1:91,1] = PR[GP1:90,1] + 40.467;
   1:  PR[GP1:91,2] = PR[GP1:90,2] + -34.469;
   1:L PR[91] 10mm/sec CNT100;
   1:  PR[GP1:91,1] = PR[GP1:90,1] + 41.655;
   1:  PR[GP1:91,2] = PR[GP1:90,2] + -34.320;
   1:L PR[91] 10mm/sec CNT100;
   1:  PR[GP1:91,1] = PR[GP1:90,1] + 47.888;
   1:  PR[GP1:91,2] = PR[GP1:90,2] + -32.019;
   1:L PR[91] 10mm/sec CNT100;
   1:  PR[GP1:91,1] = PR[GP1:90,1] + 53.198;
   1:  PR[GP1:91,2] = PR[GP1:90,2] + -30.098;
   1:L PR[91] 10mm/sec CNT100;
   1:  PR[GP1:91,1] = PR[GP1:90,1] + 54.299;
   1:  PR[GP1:91,2] = PR[GP1:90,2] + -29.242;
   1:L PR[91] 10mm/sec CNT100;
   1:  PR[GP1:91,1] = PR[GP1:90,1] + 62.662;
   1:  PR[GP1:91,2] = PR[GP1:90,2] + -22.338;
   1:L PR[91] 10mm/sec CNT100;
   1:  PR[GP1:91,1] = PR[GP1:90,1] + 64.548;
   1:  PR[GP1:91,2] = PR[GP1:90,2] + -19.262;
   1:L PR[91] 10mm/sec CNT100;
   1:  PR[GP1:91,1] = PR[GP1:90,1] + 68.942;
   1:  PR[GP1:91,2] = PR[GP1:90,2] + -11.794;
   1:L PR[91] 10mm/sec CNT100;
   1:  PR[GP1:91,1] = PR[GP1:90,1] + 69.810;
   1:  PR[GP1:91,2] = PR[GP1:90,2] + -7.146;
   1:L PR[91] 10mm/sec CNT100;
   1:  PR[GP1:91,1] = PR[GP1:90,1] + 69.912;
   1:  PR[GP1:91,2] = PR[GP1:90,2] + -6.673;
   1:L PR[91] 10mm/sec CNT100;
   1:  PR[GP1:91,1] = PR[GP1:90,1] + 71.156;
   1:  PR[GP1:91,2] = PR[GP1:90,2] + 0.276;
   1:L PR[91] 10mm/sec CNT100;
   1:  PR[GP1:91,1] = PR[GP1:90,1] + 70.217;
   1:  PR[GP1:91,2] = PR[GP1:90,2] + 5.197;
   1:L PR[91] 10mm/sec CNT100;
   1:  PR[GP1:91,1] = PR[GP1:90,1] + 68.941;
   1:  PR[GP1:91,2] = PR[GP1:90,2] + 12.355;
   1:L PR[91] 10mm/sec CNT100;
   1:  PR[GP1:91,1] = PR[GP1:90,1] + 64.548;
   1:  PR[GP1:91,2] = PR[GP1:90,2] + 19.820;
   1:L PR[91] 10mm/sec CNT100;
   1:  PR[GP1:91,1] = PR[GP1:90,1] + 62.662;
   1:  PR[GP1:91,2] = PR[GP1:90,2] + 22.896;
   1:L PR[91] 10mm/sec CNT100;
   1:  PR[GP1:91,1] = PR[GP1:90,1] + 54.299;
   1:  PR[GP1:91,2] = PR[GP1:90,2] + 29.800;
   1:L PR[91] 10mm/sec CNT100;
   1:  PR[GP1:91,1] = PR[GP1:90,1] + 53.198;
   1:  PR[GP1:91,2] = PR[GP1:90,2] + 30.656;
   1:L PR[91] 10mm/sec CNT100;
   1:  PR[GP1:91,1] = PR[GP1:90,1] + 47.888;
   1:  PR[GP1:91,2] = PR[GP1:90,2] + 32.577;
   1:L PR[91] 10mm/sec CNT100;
   1:  PR[GP1:91,1] = PR[GP1:90,1] + 41.655;
   1:  PR[GP1:91,2] = PR[GP1:90,2] + 34.878;
   1:L PR[91] 10mm/sec CNT100;
   1:  PR[GP1:91,1] = PR[GP1:90,1] + 40.467;
   1:  PR[GP1:91,2] = PR[GP1:90,2] + 35.027;
   1:L PR[91] 10mm/sec CNT100;
   1:  PR[GP1:91,1] = PR[GP1:90,1] + 30.959;
   1:  PR[GP1:91,2] = PR[GP1:90,2] + 35.305;
   1:L PR[91] 10mm/sec CNT100;
   1:  PR[GP1:91,1] = PR[GP1:90,1] + 27.828;
   1:  PR[GP1:91,2] = PR[GP1:90,2] + 35.035;
   1:L PR[91] 10mm/sec CNT100;
   1:  PR[GP1:91,1] = PR[GP1:90,1] + 22.516;
   1:  PR[GP1:91,2] = PR[GP1:90,2] + 33.334;
   1:L PR[91] 10mm/sec CNT100;
   1:  PR[GP1:91,1] = PR[GP1:90,1] + 18.245;
   1:  PR[GP1:91,2] = PR[GP1:90,2] + 32.102;
   1:L PR[91] 10mm/sec CNT100;
   1:  PR[GP1:91,1] = PR[GP1:90,1] + 12.217;
   1:  PR[GP1:91,2] = PR[GP1:90,2] + 28.686;
   1:L PR[91] 10mm/sec CNT100;
   1:  PR[GP1:91,1] = PR[GP1:90,1] + 11.495;
   1:  PR[GP1:91,2] = PR[GP1:90,2] + 28.143;
   1:L PR[91] 10mm/sec CNT100;
   1:  PR[GP1:91,1] = PR[GP1:90,1] + 9.543;
   1:  PR[GP1:91,2] = PR[GP1:90,2] + 26.384;
   1:L PR[91] 10mm/sec CNT100;
   1:  PR[GP1:91,1] = PR[GP1:90,1] + 5.844;
   1:  PR[GP1:91,2] = PR[GP1:90,2] + 23.126;
   1:L PR[91] 10mm/sec CNT100;
   1:  PR[GP1:91,1] = PR[GP1:90,1] + 5.572;
   1:  PR[GP1:91,2] = PR[GP1:90,2] + 22.795;
   1:L PR[91] 10mm/sec CNT100;
   1:  PR[GP1:91,1] = PR[GP1:90,1] + 1.460;
   1:  PR[GP1:91,2] = PR[GP1:90,2] + 17.015;
   1:L PR[91] 10mm/sec CNT100;
   1:  PR[GP1:91,1] = PR[GP1:90,1] + -1.981;
   1:L PR[91] 10mm/sec CNT100;
   1:  PR[GP1:91,1] = PR[GP1:90,1] + -6.056;
   1:  PR[GP1:91,2] = PR[GP1:90,2] + 22.761;
   1:L PR[91] 10mm/sec CNT100;
   1:  PR[GP1:91,1] = PR[GP1:90,1] + -6.325;
   1:  PR[GP1:91,2] = PR[GP1:90,2] + 23.087;
   1:L PR[91] 10mm/sec CNT100;
   1:  PR[GP1:91,1] = PR[GP1:90,1] + -10.069;
   1:  PR[GP1:91,2] = PR[GP1:90,2] + 26.384;
   1:L PR[91] 10mm/sec CNT100;
   1:  PR[GP1:91,1] = PR[GP1:90,1] + -11.995;
   1:  PR[GP1:91,2] = PR[GP1:90,2] + 28.119;
   1:L PR[91] 10mm/sec CNT100;
   1:  PR[GP1:91,1] = PR[GP1:90,1] + -12.707;
   1:  PR[GP1:91,2] = PR[GP1:90,2] + 28.655;
   1:L PR[91] 10mm/sec CNT100;
   1:  PR[GP1:91,1] = PR[GP1:90,1] + -18.785;
   1:  PR[GP1:91,2] = PR[GP1:90,2] + 32.109;
   1:L PR[91] 10mm/sec CNT100;
   1:  PR[GP1:91,1] = PR[GP1:90,1] + -23.243;
   1:  PR[GP1:91,2] = PR[GP1:90,2] + 33.516;
   1:L PR[91] 10mm/sec CNT100;
   1:  PR[GP1:91,1] = PR[GP1:90,1] + -28.350;
   1:  PR[GP1:91,2] = PR[GP1:90,2] + 35.035;
   1:L PR[91] 10mm/sec CNT100;
   1:  PR[GP1:91,1] = PR[GP1:90,1] + -31.495;
   1:  PR[GP1:91,2] = PR[GP1:90,2] + 35.305;
   1:L PR[91] 10mm/sec CNT100;
   1:  PR[GP1:91,1] = PR[GP1:90,1] + -41.002;
   1:  PR[GP1:91,2] = PR[GP1:90,2] + 35.026;
   1:L PR[91] 10mm/sec CNT100;
   1:  PR[GP1:91,1] = PR[GP1:90,1] + -42.190;
   1:  PR[GP1:91,2] = PR[GP1:90,2] + 34.877;
   1:L PR[91] 10mm/sec CNT100;
   1:  PR[GP1:91,1] = PR[GP1:90,1] + -48.414;
   1:  PR[GP1:91,2] = PR[GP1:90,2] + 32.575;
   1:L PR[91] 10mm/sec CNT100;
   1:  PR[GP1:91,1] = PR[GP1:90,1] + -53.727;
   1:  PR[GP1:91,2] = PR[GP1:90,2] + 30.651;
   1:L PR[91] 10mm/sec CNT100;
   1:  PR[GP1:91,1] = PR[GP1:90,1] + -54.829;
   1:  PR[GP1:91,2] = PR[GP1:90,2] + 29.795;
   1:L PR[91] 10mm/sec CNT100;
   1:  PR[GP1:91,1] = PR[GP1:90,1] + -63.190;
   1:  PR[GP1:91,2] = PR[GP1:90,2] + 22.901;
   1:L PR[91] 10mm/sec CNT100;
   1:  PR[GP1:91,1] = PR[GP1:90,1] + -65.075;
   1:  PR[GP1:91,2] = PR[GP1:90,2] + 19.822;
   1:L PR[91] 10mm/sec CNT100;
   1:  PR[GP1:91,1] = PR[GP1:90,1] + -69.469;
   1:  PR[GP1:91,2] = PR[GP1:90,2] + 12.334;
   1:L PR[91] 10mm/sec CNT100;
   1:  PR[GP1:91,1] = PR[GP1:90,1] + -70.337;
   1:  PR[GP1:91,2] = PR[GP1:90,2] + 7.690;
   1:L PR[91] 10mm/sec CNT100;
   1:  PR[GP1:91,1] = PR[GP1:90,1] + -70.438;
   1:  PR[GP1:91,2] = PR[GP1:90,2] + 7.218;
   1:L PR[91] 10mm/sec CNT100;
   1:  PR[GP1:91,1] = PR[GP1:90,1] + -71.682;
   1:  PR[GP1:91,2] = PR[GP1:90,2] + 0.282;
   1:L PR[91] 10mm/sec CNT100;
   1:  PR[GP1:91,1] = PR[GP1:90,1] + -70.744;
   1:  PR[GP1:91,2] = PR[GP1:90,2] + -4.634;
   1:L PR[91] 10mm/sec CNT100;
   1:  PR[GP1:91,1] = PR[GP1:90,1] + -69.468;
   1:  PR[GP1:91,2] = PR[GP1:90,2] + -11.778;
   1:L PR[91] 10mm/sec CNT100;
   1:  PR[GP1:91,1] = PR[GP1:90,1] + -65.075;
   1:  PR[GP1:91,2] = PR[GP1:90,2] + -19.264;
   1:L PR[91] 10mm/sec CNT100;
   1:  PR[GP1:91,1] = PR[GP1:90,1] + -63.190;
   1:  PR[GP1:91,2] = PR[GP1:90,2] + -22.343;
   1:L PR[91] 10mm/sec CNT100;
   1:  PR[GP1:91,1] = PR[GP1:90,1] + -54.829;
   1:  PR[GP1:91,2] = PR[GP1:90,2] + -29.237;
   1:L PR[91] 10mm/sec CNT100;
   1:  PR[GP1:91,1] = PR[GP1:90,1] + -53.727;
   1:  PR[GP1:91,2] = PR[GP1:90,2] + -30.093;
   1:L PR[91] 10mm/sec CNT100;
   1:  PR[GP1:91,1] = PR[GP1:90,1] + -48.414;
   1:  PR[GP1:91,2] = PR[GP1:90,2] + -32.017;
   1:L PR[91] 10mm/sec CNT100;
   1:  PR[GP1:91,1] = PR[GP1:90,1] + -42.190;
   1:  PR[GP1:91,2] = PR[GP1:90,2] + -34.319;
   1:L PR[91] 10mm/sec CNT100;
   1:  PR[GP1:91,1] = PR[GP1:90,1] + -41.002;
   1:  PR[GP1:91,2] = PR[GP1:90,2] + -34.468;
   1:L PR[91] 10mm/sec CNT100;
   1:  PR[GP1:91,1] = PR[GP1:90,1] + -31.495;
   1:  PR[GP1:91,2] = PR[GP1:90,2] + -34.747;
   1:L PR[91] 10mm/sec CNT100;
   1:  PR[GP1:91,1] = PR[GP1:90,1] + -28.356;
   1:  PR[GP1:91,2] = PR[GP1:90,2] + -34.478;
   1:L PR[91] 10mm/sec CNT100;
   1:  PR[GP1:91,1] = PR[GP1:90,1] + -23.044;
   1:  PR[GP1:91,2] = PR[GP1:90,2] + -32.776;
   1:L PR[91] 10mm/sec CNT100;
   1:  PR[GP1:91,1] = PR[GP1:90,1] + -18.778;
   1:  PR[GP1:91,2] = PR[GP1:90,2] + -31.547;
   1:L PR[91] 10mm/sec CNT100;
   1:  PR[GP1:91,1] = PR[GP1:90,1] + -12.707;
   1:  PR[GP1:91,2] = PR[GP1:90,2] + -28.097;
   1:L PR[91] 10mm/sec CNT100;
   1:  PR[GP1:91,1] = PR[GP1:90,1] + -11.995;
   1:  PR[GP1:91,2] = PR[GP1:90,2] + -27.561;
   1:L PR[91] 10mm/sec CNT100;
   1:  PR[GP1:91,1] = PR[GP1:90,1] + -10.069;
   1:  PR[GP1:91,2] = PR[GP1:90,2] + -25.826;
   1:L PR[91] 10mm/sec CNT100;
   1:  PR[GP1:91,1] = PR[GP1:90,1] + -6.326;
   1:  PR[GP1:91,2] = PR[GP1:90,2] + -22.531;
   1:L PR[91] 10mm/sec CNT100;
   1:  PR[GP1:91,1] = PR[GP1:90,1] + -6.058;
   1:  PR[GP1:91,2] = PR[GP1:90,2] + -22.205;
   1:L PR[91] 10mm/sec CNT100;
   1:  PR[GP1:91,1] = PR[GP1:90,1] + -1.982;
   1:  PR[GP1:91,2] = PR[GP1:90,2] + -16.457;
   1:L PR[91] 10mm/sec CNT100;
   1:  PR[GP1:91,1] = PR[GP1:90,1] + 1.461;
   1:L PR[91] 10mm/sec CNT100;
   1:  PR[GP1:91,1] = PR[GP1:90,1] + 5.146;
   1:  PR[GP1:91,2] = PR[GP1:90,2] + -22.083;
   1:  PR[GP1:91,3] = PR[GP1:90,3] + 39.345;
   1:L PR[91] 10mm/sec CNT100;
   1:  PR[GP1:91,1] = PR[GP1:90,1] + 5.618;
   1:  PR[GP1:91,2] = PR[GP1:90,2] + -22.657;
   1:L PR[91] 10mm/sec CNT100;
   1:  PR[GP1:91,1] = PR[GP1:90,1] + 11.614;
   1:  PR[GP1:91,2] = PR[GP1:90,2] + -27.937;
   1:L PR[91] 10mm/sec CNT100;
   1:  PR[GP1:91,1] = PR[GP1:90,1] + 18.224;
   1:  PR[GP1:91,2] = PR[GP1:90,2] + -31.680;
   1:L PR[91] 10mm/sec CNT100;
   1:  PR[GP1:91,1] = PR[GP1:90,1] + 21.526;
   1:  PR[GP1:91,2] = PR[GP1:90,2] + -32.722;
   1:L PR[91] 10mm/sec CNT100;
   1:  PR[GP1:91,1] = PR[GP1:90,1] + 27.485;
   1:  PR[GP1:91,2] = PR[GP1:90,2] + -34.496;
   1:L PR[91] 10mm/sec CNT100;
   1:  PR[GP1:91,1] = PR[GP1:90,1] + 31.150;
   1:  PR[GP1:91,2] = PR[GP1:90,2] + -34.811;
   1:L PR[91] 10mm/sec CNT100;
   1:  PR[GP1:91,1] = PR[GP1:90,1] + 39.759;
   1:  PR[GP1:91,2] = PR[GP1:90,2] + -34.560;
   1:L PR[91] 10mm/sec CNT100;
   1:  PR[GP1:91,1] = PR[GP1:90,1] + 41.574;
   1:  PR[GP1:91,2] = PR[GP1:90,2] + -34.332;
   1:L PR[91] 10mm/sec CNT100;
   1:  PR[GP1:91,1] = PR[GP1:90,1] + 50.878;
   1:  PR[GP1:91,2] = PR[GP1:90,2] + -30.897;
   1:L PR[91] 10mm/sec CNT100;
   1:  PR[GP1:91,1] = PR[GP1:90,1] + 53.143;
   1:  PR[GP1:91,2] = PR[GP1:90,2] + -30.078;
   1:L PR[91] 10mm/sec CNT100;
   1:  PR[GP1:91,1] = PR[GP1:90,1] + 53.577;
   1:  PR[GP1:91,2] = PR[GP1:90,2] + -29.741;
   1:L PR[91] 10mm/sec CNT100;
   1:  PR[GP1:91,1] = PR[GP1:90,1] + 62.575;
   1:  PR[GP1:91,2] = PR[GP1:90,2] + -22.312;
   1:L PR[91] 10mm/sec CNT100;
   1:  PR[GP1:91,1] = PR[GP1:90,1] + 64.064;
   1:  PR[GP1:91,2] = PR[GP1:90,2] + -19.884;
   1:L PR[91] 10mm/sec CNT100;
   1:  PR[GP1:91,1] = PR[GP1:90,1] + 68.834;
   1:  PR[GP1:91,2] = PR[GP1:90,2] + -11.778;
   1:L PR[91] 10mm/sec CNT100;
   1:  PR[GP1:91,1] = PR[GP1:90,1] + 69.573;
   1:  PR[GP1:91,2] = PR[GP1:90,2] + -7.816;
   1:L PR[91] 10mm/sec CNT100;
   1:  PR[GP1:91,1] = PR[GP1:90,1] + 69.660;
   1:  PR[GP1:91,2] = PR[GP1:90,2] + -7.412;
   1:L PR[91] 10mm/sec CNT100;
   1:  PR[GP1:91,1] = PR[GP1:90,1] + 71.037;
   1:  PR[GP1:91,2] = PR[GP1:90,2] + 0.276;
   1:L PR[91] 10mm/sec CNT100;
   1:  PR[GP1:91,1] = PR[GP1:90,1] + 70.218;
   1:  PR[GP1:91,2] = PR[GP1:90,2] + 4.568;
   1:L PR[91] 10mm/sec CNT100;
   1:  PR[GP1:91,1] = PR[GP1:90,1] + 68.832;
   1:  PR[GP1:91,2] = PR[GP1:90,2] + 12.338;
   1:L PR[91] 10mm/sec CNT100;
   1:  PR[GP1:91,1] = PR[GP1:90,1] + 64.064;
   1:  PR[GP1:91,2] = PR[GP1:90,2] + 20.442;
   1:L PR[91] 10mm/sec CNT100;
   1:  PR[GP1:91,1] = PR[GP1:90,1] + 62.575;
   1:  PR[GP1:91,2] = PR[GP1:90,2] + 22.870;
   1:L PR[91] 10mm/sec CNT100;
   1:  PR[GP1:91,1] = PR[GP1:90,1] + 53.577;
   1:  PR[GP1:91,2] = PR[GP1:90,2] + 30.299;
   1:L PR[91] 10mm/sec CNT100;
   1:  PR[GP1:91,1] = PR[GP1:90,1] + 53.144;
   1:  PR[GP1:91,2] = PR[GP1:90,2] + 30.636;
   1:L PR[91] 10mm/sec CNT100;
   1:  PR[GP1:91,1] = PR[GP1:90,1] + 50.878;
   1:  PR[GP1:91,2] = PR[GP1:90,2] + 31.455;
   1:L PR[91] 10mm/sec CNT100;
   1:  PR[GP1:91,1] = PR[GP1:90,1] + 41.574;
   1:  PR[GP1:91,2] = PR[GP1:90,2] + 34.890;
   1:L PR[91] 10mm/sec CNT100;
   1:  PR[GP1:91,1] = PR[GP1:90,1] + 39.760;
   1:  PR[GP1:91,2] = PR[GP1:90,2] + 35.118;
   1:L PR[91] 10mm/sec CNT100;
   1:  PR[GP1:91,1] = PR[GP1:90,1] + 31.150;
   1:  PR[GP1:91,2] = PR[GP1:90,2] + 35.369;
   1:L PR[91] 10mm/sec CNT100;
   1:  PR[GP1:91,1] = PR[GP1:90,1] + 27.491;
   1:  PR[GP1:91,2] = PR[GP1:90,2] + 35.054;
   1:L PR[91] 10mm/sec CNT100;
   1:  PR[GP1:91,1] = PR[GP1:90,1] + 22.924;
   1:  PR[GP1:91,2] = PR[GP1:90,2] + 33.591;
   1:L PR[91] 10mm/sec CNT100;
   1:  PR[GP1:91,1] = PR[GP1:90,1] + 18.218;
   1:  PR[GP1:91,2] = PR[GP1:90,2] + 32.234;
   1:L PR[91] 10mm/sec CNT100;
   1:  PR[GP1:91,1] = PR[GP1:90,1] + 11.617;
   1:  PR[GP1:91,2] = PR[GP1:90,2] + 28.497;
   1:L PR[91] 10mm/sec CNT100;
   1:  PR[GP1:91,1] = PR[GP1:90,1] + 5.614;
   1:  PR[GP1:91,2] = PR[GP1:90,2] + 23.212;
   1:L PR[91] 10mm/sec CNT100;
   1:  PR[GP1:91,1] = PR[GP1:90,1] + 5.135;
   1:  PR[GP1:91,2] = PR[GP1:90,2] + 22.627;
   1:L PR[91] 10mm/sec CNT100;
   1:  PR[GP1:91,1] = PR[GP1:90,1] + 1.374;
   1:  PR[GP1:91,2] = PR[GP1:90,2] + 17.340;
   1:L PR[91] 10mm/sec CNT100;
   1:  PR[GP1:91,1] = PR[GP1:90,1] + -1.894;
   1:L PR[91] 10mm/sec CNT100;
   1:  PR[GP1:91,1] = PR[GP1:90,1] + -5.624;
   1:  PR[GP1:91,2] = PR[GP1:90,2] + 22.600;
   1:L PR[91] 10mm/sec CNT100;
   1:  PR[GP1:91,1] = PR[GP1:90,1] + -6.097;
   1:  PR[GP1:91,2] = PR[GP1:90,2] + 23.174;
   1:L PR[91] 10mm/sec CNT100;
   1:  PR[GP1:91,1] = PR[GP1:90,1] + -12.110;
   1:  PR[GP1:91,2] = PR[GP1:90,2] + 28.467;
   1:L PR[91] 10mm/sec CNT100;
   1:  PR[GP1:91,1] = PR[GP1:90,1] + -18.758;
   1:  PR[GP1:91,2] = PR[GP1:90,2] + 32.241;
   1:L PR[91] 10mm/sec CNT100;
   1:  PR[GP1:91,1] = PR[GP1:90,1] + -22.062;
   1:  PR[GP1:91,2] = PR[GP1:90,2] + 33.284;
   1:L PR[91] 10mm/sec CNT100;
   1:  PR[GP1:91,1] = PR[GP1:90,1] + -28.012;
   1:  PR[GP1:91,2] = PR[GP1:90,2] + 35.055;
   1:L PR[91] 10mm/sec CNT100;
   1:  PR[GP1:91,1] = PR[GP1:90,1] + -31.687;
   1:  PR[GP1:91,2] = PR[GP1:90,2] + 35.369;
   1:L PR[91] 10mm/sec CNT100;
   1:  PR[GP1:91,1] = PR[GP1:90,1] + -40.296;
   1:  PR[GP1:91,2] = PR[GP1:90,2] + 35.117;
   1:L PR[91] 10mm/sec CNT100;
   1:  PR[GP1:91,1] = PR[GP1:90,1] + -42.112;
   1:  PR[GP1:91,2] = PR[GP1:90,2] + 34.888;
   1:L PR[91] 10mm/sec CNT100;
   1:  PR[GP1:91,1] = PR[GP1:90,1] + -51.404;
   1:  PR[GP1:91,2] = PR[GP1:90,2] + 31.452;
   1:L PR[91] 10mm/sec CNT100;
   1:  PR[GP1:91,1] = PR[GP1:90,1] + -53.673;
   1:  PR[GP1:91,2] = PR[GP1:90,2] + 30.631;
   1:L PR[91] 10mm/sec CNT100;
   1:  PR[GP1:91,1] = PR[GP1:90,1] + -54.108;
   1:  PR[GP1:91,2] = PR[GP1:90,2] + 30.293;
   1:L PR[91] 10mm/sec CNT100;
   1:  PR[GP1:91,1] = PR[GP1:90,1] + -63.103;
   1:  PR[GP1:91,2] = PR[GP1:90,2] + 22.876;
   1:L PR[91] 10mm/sec CNT100;
   1:  PR[GP1:91,1] = PR[GP1:90,1] + -64.591;
   1:  PR[GP1:91,2] = PR[GP1:90,2] + 20.445;
   1:L PR[91] 10mm/sec CNT100;
   1:  PR[GP1:91,1] = PR[GP1:90,1] + -69.360;
   1:  PR[GP1:91,2] = PR[GP1:90,2] + 12.317;
   1:L PR[91] 10mm/sec CNT100;
   1:  PR[GP1:91,1] = PR[GP1:90,1] + -70.100;
   1:  PR[GP1:91,2] = PR[GP1:90,2] + 8.359;
   1:L PR[91] 10mm/sec CNT100;
   1:  PR[GP1:91,1] = PR[GP1:90,1] + -70.187;
   1:  PR[GP1:91,2] = PR[GP1:90,2] + 7.956;
   1:L PR[91] 10mm/sec CNT100;
   1:  PR[GP1:91,1] = PR[GP1:90,1] + -71.563;
   1:  PR[GP1:91,2] = PR[GP1:90,2] + 0.282;
   1:L PR[91] 10mm/sec CNT100;
   1:  PR[GP1:91,1] = PR[GP1:90,1] + -70.745;
   1:  PR[GP1:91,2] = PR[GP1:90,2] + -4.006;
   1:L PR[91] 10mm/sec CNT100;
   1:  PR[GP1:91,1] = PR[GP1:90,1] + -69.359;
   1:  PR[GP1:91,2] = PR[GP1:90,2] + -11.761;
   1:L PR[91] 10mm/sec CNT100;
   1:  PR[GP1:91,1] = PR[GP1:90,1] + -64.591;
   1:  PR[GP1:91,2] = PR[GP1:90,2] + -19.887;
   1:L PR[91] 10mm/sec CNT100;
   1:  PR[GP1:91,1] = PR[GP1:90,1] + -63.103;
   1:  PR[GP1:91,2] = PR[GP1:90,2] + -22.318;
   1:L PR[91] 10mm/sec CNT100;
   1:  PR[GP1:91,1] = PR[GP1:90,1] + -54.108;
   1:  PR[GP1:91,2] = PR[GP1:90,2] + -29.735;
   1:L PR[91] 10mm/sec CNT100;
   1:  PR[GP1:91,1] = PR[GP1:90,1] + -53.673;
   1:  PR[GP1:91,2] = PR[GP1:90,2] + -30.073;
   1:L PR[91] 10mm/sec CNT100;
   1:  PR[GP1:91,1] = PR[GP1:90,1] + -51.404;
   1:  PR[GP1:91,2] = PR[GP1:90,2] + -30.894;
   1:L PR[91] 10mm/sec CNT100;
   1:  PR[GP1:91,1] = PR[GP1:90,1] + -42.112;
   1:  PR[GP1:91,2] = PR[GP1:90,2] + -34.330;
   1:L PR[91] 10mm/sec CNT100;
   1:  PR[GP1:91,1] = PR[GP1:90,1] + -40.296;
   1:  PR[GP1:91,2] = PR[GP1:90,2] + -34.559;
   1:L PR[91] 10mm/sec CNT100;
   1:  PR[GP1:91,1] = PR[GP1:90,1] + -31.687;
   1:  PR[GP1:91,2] = PR[GP1:90,2] + -34.811;
   1:L PR[91] 10mm/sec CNT100;
   1:  PR[GP1:91,1] = PR[GP1:90,1] + -28.019;
   1:  PR[GP1:91,2] = PR[GP1:90,2] + -34.497;
   1:L PR[91] 10mm/sec CNT100;
   1:  PR[GP1:91,1] = PR[GP1:90,1] + -23.451;
   1:  PR[GP1:91,2] = PR[GP1:90,2] + -33.034;
   1:L PR[91] 10mm/sec CNT100;
   1:  PR[GP1:91,1] = PR[GP1:90,1] + -18.751;
   1:  PR[GP1:91,2] = PR[GP1:90,2] + -31.679;
   1:L PR[91] 10mm/sec CNT100;
   1:  PR[GP1:91,1] = PR[GP1:90,1] + -12.106;
   1:  PR[GP1:91,2] = PR[GP1:90,2] + -27.906;
   1:L PR[91] 10mm/sec CNT100;
   1:  PR[GP1:91,1] = PR[GP1:90,1] + -6.100;
   1:  PR[GP1:91,2] = PR[GP1:90,2] + -22.620;
   1:L PR[91] 10mm/sec CNT100;
   1:  PR[GP1:91,1] = PR[GP1:90,1] + -5.628;
   1:  PR[GP1:91,2] = PR[GP1:90,2] + -22.046;
   1:L PR[91] 10mm/sec CNT100;
   1:  PR[GP1:91,1] = PR[GP1:90,1] + -1.895;
   1:  PR[GP1:91,2] = PR[GP1:90,2] + -16.782;
   1:L PR[91] 10mm/sec CNT100;
   1:  PR[GP1:91,1] = PR[GP1:90,1] + 1.375;
   1:L PR[91] 10mm/sec CNT100;
   1:  PR[GP1:91,1] = PR[GP1:90,1] + 4.713;
   1:  PR[GP1:91,2] = PR[GP1:90,2] + -21.920;
   1:  PR[GP1:91,3] = PR[GP1:90,3] + 39.955;
   1:L PR[91] 10mm/sec CNT100;
   1:  PR[GP1:91,1] = PR[GP1:90,1] + 5.390;
   1:  PR[GP1:91,2] = PR[GP1:90,2] + -22.744;
   1:L PR[91] 10mm/sec CNT100;
   1:  PR[GP1:91,1] = PR[GP1:90,1] + 11.365;
   1:  PR[GP1:91,2] = PR[GP1:90,2] + -28.002;
   1:L PR[91] 10mm/sec CNT100;
   1:  PR[GP1:91,1] = PR[GP1:90,1] + 13.909;
   1:  PR[GP1:91,2] = PR[GP1:90,2] + -29.383;
   1:L PR[91] 10mm/sec CNT100;
   1:  PR[GP1:91,1] = PR[GP1:90,1] + 18.197;
   1:  PR[GP1:91,2] = PR[GP1:90,2] + -31.812;
   1:L PR[91] 10mm/sec CNT100;
   1:  PR[GP1:91,1] = PR[GP1:90,1] + 20.344;
   1:  PR[GP1:91,2] = PR[GP1:90,2] + -32.490;
   1:L PR[91] 10mm/sec CNT100;
   1:  PR[GP1:91,1] = PR[GP1:90,1] + 27.148;
   1:  PR[GP1:91,2] = PR[GP1:90,2] + -34.515;
   1:L PR[91] 10mm/sec CNT100;
   1:  PR[GP1:91,1] = PR[GP1:90,1] + 31.341;
   1:  PR[GP1:91,2] = PR[GP1:90,2] + -34.876;
   1:L PR[91] 10mm/sec CNT100;
   1:  PR[GP1:91,1] = PR[GP1:90,1] + 39.052;
   1:  PR[GP1:91,2] = PR[GP1:90,2] + -34.651;
   1:L PR[91] 10mm/sec CNT100;
   1:  PR[GP1:91,1] = PR[GP1:90,1] + 41.494;
   1:  PR[GP1:91,2] = PR[GP1:90,2] + -34.345;
   1:L PR[91] 10mm/sec CNT100;
   1:  PR[GP1:91,1] = PR[GP1:90,1] + 53.053;
   1:  PR[GP1:91,2] = PR[GP1:90,2] + -30.077;
   1:L PR[91] 10mm/sec CNT100;
   1:  PR[GP1:91,1] = PR[GP1:90,1] + 53.060;
   1:  PR[GP1:91,2] = PR[GP1:90,2] + -30.073;
   1:L PR[91] 10mm/sec CNT100;
   1:  PR[GP1:91,1] = PR[GP1:90,1] + 62.488;
   1:  PR[GP1:91,2] = PR[GP1:90,2] + -22.286;
   1:L PR[91] 10mm/sec CNT100;
   1:  PR[GP1:91,1] = PR[GP1:90,1] + 63.580;
   1:  PR[GP1:91,2] = PR[GP1:90,2] + -20.506;
   1:L PR[91] 10mm/sec CNT100;
   1:  PR[GP1:91,1] = PR[GP1:90,1] + 68.725;
   1:  PR[GP1:91,2] = PR[GP1:90,2] + -11.761;
   1:L PR[91] 10mm/sec CNT100;
   1:  PR[GP1:91,1] = PR[GP1:90,1] + 69.407;
   1:  PR[GP1:91,2] = PR[GP1:90,2] + -8.158;
   1:L PR[91] 10mm/sec CNT100;
   1:  PR[GP1:91,1] = PR[GP1:90,1] + 70.918;
   1:  PR[GP1:91,2] = PR[GP1:90,2] + 0.276;
   1:L PR[91] 10mm/sec CNT100;
   1:  PR[GP1:91,1] = PR[GP1:90,1] + 70.219;
   1:  PR[GP1:91,2] = PR[GP1:90,2] + 3.939;
   1:L PR[91] 10mm/sec CNT100;
   1:  PR[GP1:91,1] = PR[GP1:90,1] + 68.724;
   1:  PR[GP1:91,2] = PR[GP1:90,2] + 12.322;
   1:L PR[91] 10mm/sec CNT100;
   1:  PR[GP1:91,1] = PR[GP1:90,1] + 63.580;
   1:  PR[GP1:91,2] = PR[GP1:90,2] + 21.064;
   1:L PR[91] 10mm/sec CNT100;
   1:  PR[GP1:91,1] = PR[GP1:90,1] + 62.488;
   1:  PR[GP1:91,2] = PR[GP1:90,2] + 22.844;
   1:L PR[91] 10mm/sec CNT100;
   1:  PR[GP1:91,1] = PR[GP1:90,1] + 53.060;
   1:  PR[GP1:91,2] = PR[GP1:90,2] + 30.631;
   1:L PR[91] 10mm/sec CNT100;
   1:  PR[GP1:91,1] = PR[GP1:90,1] + 53.053;
   1:  PR[GP1:91,2] = PR[GP1:90,2] + 30.635;
   1:L PR[91] 10mm/sec CNT100;
   1:  PR[GP1:91,1] = PR[GP1:90,1] + 43.016;
   1:  PR[GP1:91,2] = PR[GP1:90,2] + 34.352;
   1:L PR[91] 10mm/sec CNT100;
   1:  PR[GP1:91,1] = PR[GP1:90,1] + 41.496;
   1:  PR[GP1:91,2] = PR[GP1:90,2] + 34.902;
   1:L PR[91] 10mm/sec CNT100;
   1:  PR[GP1:91,1] = PR[GP1:90,1] + 39.052;
   1:  PR[GP1:91,2] = PR[GP1:90,2] + 35.209;
   1:L PR[91] 10mm/sec CNT100;
   1:  PR[GP1:91,1] = PR[GP1:90,1] + 31.341;
   1:  PR[GP1:91,2] = PR[GP1:90,2] + 35.434;
   1:L PR[91] 10mm/sec CNT100;
   1:  PR[GP1:91,1] = PR[GP1:90,1] + 27.155;
   1:  PR[GP1:91,2] = PR[GP1:90,2] + 35.073;
   1:L PR[91] 10mm/sec CNT100;
   1:  PR[GP1:91,1] = PR[GP1:90,1] + 23.331;
   1:  PR[GP1:91,2] = PR[GP1:90,2] + 33.849;
   1:L PR[91] 10mm/sec CNT100;
   1:  PR[GP1:91,1] = PR[GP1:90,1] + 18.190;
   1:  PR[GP1:91,2] = PR[GP1:90,2] + 32.366;
   1:L PR[91] 10mm/sec CNT100;
   1:  PR[GP1:91,1] = PR[GP1:90,1] + 13.909;
   1:  PR[GP1:91,2] = PR[GP1:90,2] + 29.940;
   1:L PR[91] 10mm/sec CNT100;
   1:  PR[GP1:91,1] = PR[GP1:90,1] + 11.429;
   1:  PR[GP1:91,2] = PR[GP1:90,2] + 28.602;
   1:L PR[91] 10mm/sec CNT100;
   1:  PR[GP1:91,1] = PR[GP1:90,1] + 11.156;
   1:  PR[GP1:91,2] = PR[GP1:90,2] + 28.379;
   1:L PR[91] 10mm/sec CNT100;
   1:  PR[GP1:91,1] = PR[GP1:90,1] + 5.385;
   1:  PR[GP1:91,2] = PR[GP1:90,2] + 23.297;
   1:L PR[91] 10mm/sec CNT100;
   1:  PR[GP1:91,1] = PR[GP1:90,1] + 4.697;
   1:  PR[GP1:91,2] = PR[GP1:90,2] + 22.458;
   1:L PR[91] 10mm/sec CNT100;
   1:  PR[GP1:91,1] = PR[GP1:90,1] + 1.287;
   1:  PR[GP1:91,2] = PR[GP1:90,2] + 17.665;
   1:L PR[91] 10mm/sec CNT100;
   1:  PR[GP1:91,1] = PR[GP1:90,1] + -1.808;
   1:L PR[91] 10mm/sec CNT100;
   1:  PR[GP1:91,1] = PR[GP1:90,1] + -5.193;
   1:  PR[GP1:91,2] = PR[GP1:90,2] + 22.439;
   1:L PR[91] 10mm/sec CNT100;
   1:  PR[GP1:91,1] = PR[GP1:90,1] + -5.870;
   1:  PR[GP1:91,2] = PR[GP1:90,2] + 23.261;
   1:L PR[91] 10mm/sec CNT100;
   1:  PR[GP1:91,1] = PR[GP1:90,1] + -11.646;
   1:  PR[GP1:91,2] = PR[GP1:90,2] + 28.347;
   1:L PR[91] 10mm/sec CNT100;
   1:  PR[GP1:91,1] = PR[GP1:90,1] + -11.923;
   1:  PR[GP1:91,2] = PR[GP1:90,2] + 28.572;
   1:L PR[91] 10mm/sec CNT100;
   1:  PR[GP1:91,1] = PR[GP1:90,1] + -14.436;
   1:  PR[GP1:91,2] = PR[GP1:90,2] + 29.933;
   1:L PR[91] 10mm/sec CNT100;
